  MoveL 756 to (-578.4, 950, 50) mm, rotated rx -180 ry 0 rz 90 deg; joints [-3.759, -80.624, 132.574, 175.231, 52.046, -177.063]
  MoveL 757 to (-578.4, 1000, 50) mm, rotated rx -180 ry 0 rz 90 deg; joints [-3.916, -82.713, 135.158, 175.065, 52.548, -176.994]
  MoveL 758 to (-578.4, 1000, -0.5) mm, rotated rx -180 ry 0 rz 90 deg; joints [-3.916, -79.629, 135.588, 175.277, 56.049, -177.358]
  MoveL 759 to (-578.4, 1000, 50) mm, rotated rx -180 ry 0 rz 90 deg; joints [-3.916, -82.713, 135.158, 175.065, 52.548, -176.994]
  MoveL 760 to (-578.4, 1050, 50) mm, rotated rx -180 ry 0 rz 90 deg; joints [-4.087, -84.881, 137.714, 174.876, 52.943, -176.907]
  MoveL 761 to (-578.4, 1050, -0.5) mm, rotated rx 180 ry 0 rz 90 deg; joints [-4.087, -81.618, 138.166, 175.105, 56.644, -177.304]
  MoveL 762 to (-578.4, 1050, 50) mm, rotated rx -180 ry 0 rz 90 deg; joints [-4.087, -84.881, 137.714, 174.876, 52.943, -176.907]
  MoveL 763 to (-578.4, 1100, 50) mm, rotated rx 180 ry 0 rz 90 deg; joints [-4.273, -87.147, 140.242, 174.661, 53.214, -176.797]
  MoveL 764 to (-578.4, 1100, -0.5) mm, rotated rx -180 ry 0 rz 90 deg; joints [-4.273, -83.684, 140.72, 174.91, 57.139, -177.233]
  MoveL 765 to (-578.4, 1100, 50) mm, rotated rx 180 ry 0 rz 90 deg; joints [-4.273, -87.147, 140.242, 174.661, 53.214, -176.797]
  MoveL 766 to (-578.4, 1150, 50) mm, rotated rx 180 ry 0 rz 90 deg; joints [-4.478, -89.533, 142.744, 174.415, 53.341, -176.659]
  MoveL 767 to (-578.4, 1150, -0.5) mm, rotated rx -180 ry 0 rz 90 deg; joints [-4.478, -85.847, 143.251, 174.69, 57.516, -177.142]
  MoveL 768 to (-578.4, 1150, 50) mm, rotated rx 180 ry 0 rz 90 deg; joints [-4.478, -89.533, 142.744, 174.415, 53.341, -176.659]
  MoveL 769 to (-578.4, 1200, 50) mm, rotated rx 180 ry 0 rz 90 deg; joints [-4.702, -92.068, 145.219, 174.131, 53.295, -176.484]
  MoveL 770 to (-578.4, 1200, -0.5) mm, rotated rx -180 ry 0 rz 90 deg; joints [-4.702, -88.13, 145.761, 174.437, 57.753, -177.025]
  MoveL 771 to (-578.4, 1200, 50) mm, rotated rx 180 ry 0 rz 90 deg; joints [-4.702, -92.068, 145.219, 174.131, 53.295, -176.484]
  MoveL 772 to (-578.4, 1250, 50) mm, rotated rx 180 ry 0 rz 90 deg; joints [-4.951, -94.787, 147.667, 173.8, 53.041, -176.263]
  MoveL 773 to (-578.4, 1250, -0.5) mm, rotated rx -180 ry 0 rz 90 deg; joints [-4.951, -90.565, 148.248, 174.148, 57.818, -176.875]
  MoveL 774 to (-578.4, 1250, 50) mm, rotated rx 180 ry 0 rz 90 deg; joints [-4.951, -94.787, 147.667, 173.8, 53.041, -176.263]
  MoveL 775 to (-578.4, 1300, 50) mm, rotated rx 180 ry 0 rz 90 deg; joints [-5.227, -97.739, 150.087, 173.409, 52.531, -175.979]
  MoveL 776 to (-578.4, 1300, -0.5) mm, rotated rx 180 ry 0 rz 90 deg; joints [-5.227, -93.195, 150.715, 173.811, 57.672, -176.681]
  MoveL 777 to (-578.4, 1300, 50) mm, rotated rx 180 ry 0 rz 90 deg; joints [-5.227, -97.739, 150.087, 173.409, 52.531, -175.979]
  MoveL 778 to (-578.4, 1350, 50) mm, rotated rx 180 ry 0 rz 90 deg; joints [-5.535, -100.986, 152.476, 172.94, 51.702, -175.611]
  MoveL 779 to (-578.4, 1350, -0.5) mm, rotated rx -180 ry 0 rz 90 deg; joints [-5.535, -96.076, 153.16, 173.415, 57.257, -176.427]
  MoveL 780 to (-578.4, 1350, 50) mm, rotated rx 180 ry 0 rz 90 deg; joints [-5.535, -100.986, 152.476, 172.94, 51.702, -175.611]
  MoveL 781 to (-578.4, 1400, 50) mm, rotated rx 180 ry 0 rz 90 deg; joints [-5.882, -104.615, 154.831, 172.364, 50.467, -175.122]
  MoveL 782 to (-578.4, 1400, -0.5) mm, rotated rx -180 ry 0 rz 70 deg; joints [-12.877, -96.991, 153.881, 142.344, 62.693, -160.506]
  MoveL 783 to (-578.4, 1400, 50) mm, rotated rx 180 ry 0 rz 90 deg; joints [-5.882, -104.615, 154.831, 172.364, 50.467, -175.122]
  MoveL 784 to (-578.4, 1450, 50) mm, rotated rx -180 ry 0 rz 50 deg; joints [-18.777, -100.129, 151.872, 115.454, 71.278, -146.007]
  MoveL 785 to (-578.4, 1450, -0.5) mm, rotated rx 180 ry 0 rz 50 deg; joints [-18.777, -95.317, 152.541, 117.006, 73.703, -151.163]
  MoveL 786 to (-578.4, 1450, 50) mm, rotated rx -180 ry 0 rz 50 deg; joints [-18.777, -100.129, 151.872, 115.454, 71.278, -146.007]
  MoveL 787 to (-514.2, 300, 50) mm, rotated rx -180 ry 0 rz 90 deg; joints [-4.407, -56.021, 95.158, 173.039, 39.345, -174.606]
  MoveL 788 to (-514.2, 300, -0.5) mm, rotated rx -180 ry 0 rz 90 deg; joints [-4.407, -54.32, 95.452, 173.318, 41.325, -174.972]
  MoveL 789 to (-514.2, 300, 50) mm, rotated rx -180 ry 0 rz 90 deg; joints [-4.407, -56.021, 95.158, 173.039, 39.345, -174.606]
  MoveL 790 to (-514.2, 650, 50) mm, rotated rx -180 ry 0 rz 90 deg; joints [-5.401, -68.907, 116.122, 172.659, 47.45, -175.021]
  MoveL 791 to (-514.2, 650, -0.5) mm, rotated rx 180 ry 0 rz 90 deg; joints [-5.401, -66.704, 116.453, 172.938, 49.963, -175.444]
  MoveL 792 to (-514.2, 650, 50) mm, rotated rx -180 ry 0 rz 90 deg; joints [-5.401, -68.907, 116.122, 172.659, 47.45, -175.021]
  MoveL 793 to (-476, 230, 50) mm, rotated rx -180 ry 0 rz 90 deg; joints [-5.358, -53.228, 90.342, 171.166, 37.444, -172.965]
  MoveL 794 to (-476, 230, -0.5) mm, rotated rx 180 ry 0 rz 90 deg; joints [-5.358, -51.608, 90.634, 171.529, 39.333, -173.429]
  MoveL 795 to (-476, 230, 50) mm, rotated rx -180 ry 0 rz 90 deg; joints [-5.358, -53.228, 90.342, 171.166, 37.444, -172.965]
  MoveL 796 to (-514.2, 230, 50) mm, rotated rx 180 ry 0 rz 90 deg; joints [-4.25, -53.352, 90.557, 172.994, 37.412, -174.425]
  MoveL 797 to (-514.2, 230, -0.5) mm, rotated rx 180 ry 0 rz 90 deg; joints [-4.25, -51.729, 90.849, 173.283, 39.314, -174.793]
  MoveL 798 to (-514.2, 230, 50) mm, rotated rx 180 ry 0 rz 90 deg; joints [-4.25, -53.352, 90.557, 172.994, 37.412, -174.425]
  MoveL 799 to (-552.4, 230, 50) mm, rotated rx -180 ry 0 rz 90 deg; joints [-3.139, -53.447, 90.723, 174.826, 37.388, -175.885]
  MoveL 800 to (-552.4, 230, -0.5) mm, rotated rx -180 ry 0 rz 90 deg; joints [-3.139, -51.821, 91.014, 175.04, 39.298, -176.158]
  MoveL 801 to (-552.4, 230, 50) mm, rotated rx -180 ry 0 rz 90 deg; joints [-3.139, -53.447, 90.723, 174.826, 37.388, -175.885]
  MoveL 802 to (-476, 420, 50) mm, rotated rx -180 ry 0 rz 90 deg; joints [-5.928, -60.356, 102.467, 171.198, 42.448, -173.481]
  MoveL 803 to (-476, 420, -0.5) mm, rotated rx -180 ry 0 rz 90 deg; joints [-5.928, -58.514, 102.768, 171.537, 44.568, -173.949]
  MoveL 804 to (-476, 420, 50) mm, rotated rx -180 ry 0 rz 90 deg; joints [-5.928, -60.356, 102.467, 171.198, 42.448, -173.481]
  MoveL 805 to (-514.2, 420, 50) mm, rotated rx -180 ry 0 rz 90 deg; joints [-4.704, -60.487, 102.684, 173.016, 42.409, -174.832]
  MoveL 806 to (-514.2, 420, -0.5) mm, rotated rx 180 ry 0 rz 90 deg; joints [-4.704, -58.64, 102.985, 173.286, 44.542, -175.204]
  MoveL 807 to (-514.2, 420, 50) mm, rotated rx -180 ry 0 rz 90 deg; joints [-4.704, -60.487, 102.684, 173.016, 42.409, -174.832]
  MoveL 808 to (-552.4, 420, 50) mm, rotated rx 180 ry 0 rz 90 deg; joints [-3.475, -60.588, 102.85, 174.841, 42.378, -176.184]
  MoveL 809 to (-552.4, 420, -0.5) mm, rotated rx -180 ry 0 rz 90 deg; joints [-3.475, -58.737, 103.152, 175.041, 44.523, -176.46]
  MoveL 810 to (-552.4, 420, 50) mm, rotated rx 180 ry 0 rz 90 deg; joints [-3.475, -60.588, 102.85, 174.841, 42.378, -176.184]
  MoveL 811 to (-476, 1020, 50) mm, rotated rx -180 ry 0 rz 90 deg; joints [-8.922, -83.074, 135.592, 168.809, 53.048, -173.218]
  MoveL 812 to (-476, 1020, -0.5) mm, rotated rx -180 ry 0 rz 90 deg; joints [-8.922, -79.961, 136.026, 169.285, 56.53, -174.042]
  MoveL 813 to (-476, 1020, 50) mm, rotated rx -180 ry 0 rz 90 deg; joints [-8.922, -83.074, 135.592, 168.809, 53.048, -173.218]
  MoveL 814 to (-514.2, 1020, 50) mm, rotated rx -180 ry 0 rz 90 deg; joints [-7.091, -83.302, 135.865, 171.096, 52.898, -174.601]
  MoveL 815 to (-514.2, 1020, -0.5) mm, rotated rx 180 ry 0 rz 90 deg; joints [-7.091, -80.171, 136.302, 171.479, 56.424, -175.263]
  MoveL 816 to (-514.2, 1020, 50) mm, rotated rx -180 ry 0 rz 90 deg; joints [-7.091, -83.302, 135.865, 171.096, 52.898, -174.601]
  MoveL 817 to (-552.4, 1020, 50) mm, rotated rx -180 ry 0 rz 90 deg; joints [-5.246, -83.479, 136.076, 173.407, 52.78, -176.001]
  MoveL 818 to (-552.4, 1020, -0.5) mm, rotated rx -180 ry 0 rz 90 deg; joints [-5.246, -80.334, 136.514, 173.694, 56.341, -176.495]
  MoveL 819 to (-552.4, 1020, 50) mm, rotated rx -180 ry 0 rz 90 deg; joints [-5.246, -83.479, 136.076, 173.407, 52.78, -176.001]
  MoveL 820 to (-655, 50, 50) mm, rotated rx -180 ry 0 rz 90 deg; joints [-0.134, -46.338, 78.157, 179.746, 31.82, -179.784]
  MoveL 821 to (-655, 50, -0.5) mm, rotated rx 180 ry 0 rz 90 deg; joints [-0.134, -44.886, 78.453, 179.758, 33.567, -179.798]
  MoveL 822 to (-655, 50, 50) mm, rotated rx -180 ry 0 rz 90 deg; joints [-0.134, -46.338, 78.157, 179.746, 31.82, -179.784]
  MoveL 823 to (-655, 100, 50) mm, rotated rx 180 ry 0 rz 90 deg; joints [-0.137, -48.409, 81.86, 179.752, 33.452, -179.793]
  MoveL 824 to (-655, 100, -0.5) mm, rotated rx -180 ry 0 rz 90 deg; joints [-0.137, -46.911, 82.153, 179.763, 35.243, -179.806]
  MoveL 825 to (-655, 100, 50) mm, rotated rx 180 ry 0 rz 90 deg; joints [-0.137, -48.409, 81.86, 179.752, 33.452, -179.793]
  MoveL 826 to (-655, 150, 50) mm, rotated rx -180 ry 0 rz 90 deg; joints [-0.14, -50.425, 85.434, 179.755, 35.009, -179.8]
  MoveL 827 to (-655, 150, -0.5) mm, rotated rx 180 ry 0 rz 90 deg; joints [-0.14, -48.879, 85.726, 179.766, 36.847, -179.813]
  MoveL 828 to (-655, 150, 50) mm, rotated rx -180 ry 0 rz 90 deg; joints [-0.14, -50.425, 85.434, 179.755, 35.009, -179.8]
  MoveL 829 to (-655, 200, 50) mm, rotated rx 180 ry 0 rz 90 deg; joints [-0.144, -52.397, 88.893, 179.758, 36.497, -179.806]
  MoveL 830 to (-655, 200, -0.5) mm, rotated rx -180 ry 0 rz 90 deg; joints [-0.144, -50.799, 89.185, 179.768, 38.386, -179.818]
  MoveL 831 to (-655, 200, 50) mm, rotated rx 180 ry 0 rz 90 deg; joints [-0.144, -52.397, 88.893, 179.758, 36.497, -179.806]
  MoveL 832 to (-655, 250, 50) mm, rotated rx 180 ry 0 rz 90 deg; joints [-0.148, -54.33, 92.252, 179.76, 37.922, -179.811]
  MoveL 833 to (-655, 250, -0.5) mm, rotated rx 180 ry 0 rz 90 deg; joints [-0.148, -52.679, 92.544, 179.77, 39.865, -179.823]
  MoveL 834 to (-655, 250, 50) mm, rotated rx 180 ry 0 rz 90 deg; joints [-0.148, -54.33, 92.252, 179.76, 37.922, -179.811]
  MoveL 835 to (-655, 300, 50) mm, rotated rx -180 ry 0 rz 90 deg; joints [-0.151, -56.232, 95.52, 179.761, 39.288, -179.815]
  MoveL 836 to (-655, 300, -0.5) mm, rotated rx 180 ry 0 rz 90 deg; joints [-0.151, -54.526, 95.814, 179.771, 41.289, -179.828]
  MoveL 837 to (-655, 300, 50) mm, rotated rx -180 ry 0 rz 90 deg; joints [-0.151, -56.232, 95.52, 179.761, 39.288, -179.815]
  MoveL 838 to (-655, 350, 50) mm, rotated rx 180 ry 0 rz 90 deg; joints [-0.156, -58.11, 98.708, 179.761, 40.598, -179.819]
  MoveL 839 to (-655, 350, -0.5) mm, rotated rx 180 ry 0 rz 90 deg; joints [-0.156, -56.344, 99.005, 179.77, 42.661, -179.831]
  MoveL 840 to (-655, 350, 50) mm, rotated rx 180 ry 0 rz 90 deg; joints [-0.156, -58.11, 98.708, 179.761, 40.598, -179.819]
  MoveL 841 to (-655, 400, 50) mm, rotated rx 180 ry 0 rz 90 deg; joints [-0.16, -59.969, 101.822, 179.76, 41.854, -179.822]
  MoveL 842 to (-655, 400, -0.5) mm, rotated rx -180 ry 0 rz 90 deg; joints [-0.16, -58.14, 102.123, 179.77, 43.983, -179.834]
  MoveL 843 to (-655, 400, 50) mm, rotated rx 180 ry 0 rz 90 deg; joints [-0.16, -59.969, 101.822, 179.76, 41.854, -179.822]
  MoveL 844 to (-655, 450, 50) mm, rotated rx 180 ry 0 rz 90 deg; joints [-0.164, -61.814, 104.871, 179.759, 43.057, -179.824]
  MoveL 845 to (-655, 450, -0.5) mm, rotated rx -180 ry 0 rz 90 deg; joints [-0.164, -59.918, 105.176, 179.768, 45.258, -179.837]
  MoveL 846 to (-655, 450, 50) mm, rotated rx 180 ry 0 rz 90 deg; joints [-0.164, -61.814, 104.871, 179.759, 43.057, -179.824]
  MoveL 847 to (-655, 500, 50) mm, rotated rx 180 ry 0 rz 90 deg; joints [-0.169, -63.65, 107.859, 179.757, 44.209, -179.826]
  MoveL 848 to (-655, 500, -0.5) mm, rotated rx -180 ry 0 rz 90 deg; joints [-0.169, -61.683, 108.169, 179.767, 46.487, -179.839]
  MoveL 849 to (-655, 500, 50) mm, rotated rx 180 ry 0 rz 90 deg; joints [-0.169, -63.65, 107.859, 179.757, 44.209, -179.826]
  MoveL 850 to (-655, 550, 50) mm, rotated rx 180 ry 0 rz 90 deg; joints [-0.174, -65.483, 110.791, 179.755, 45.309, -179.827]
  MoveL 851 to (-655, 550, -0.5) mm, rotated rx 180 ry 0 rz 90 deg; joints [-0.174, -63.439, 111.108, 179.764, 47.669, -179.841]
  MoveL 852 to (-655, 550, 50) mm, rotated rx 180 ry 0 rz 90 deg; joints [-0.174, -65.483, 110.791, 179.755, 45.309, -179.827]
  MoveL 853 to (-655, 600, 50) mm, rotated rx -180 ry 0 rz 90 deg; joints [-0.18, -67.318, 113.673, 179.751, 46.356, -179.828]
  MoveL 854 to (-655, 600, -0.5) mm, rotated rx 180 ry 0 rz 90 deg; joints [-0.18, -65.192, 113.997, 179.761, 48.806, -179.842]
  MoveL 855 to (-655, 600, 50) mm, rotated rx -180 ry 0 rz 90 deg; joints [-0.18, -67.318, 113.673, 179.751, 46.356, -179.828]
  MoveL 856 to (-655, 650, 50) mm, rotated rx 180 ry 0 rz 90 deg; joints [-0.186, -69.16, 116.509, 179.747, 47.349, -179.829]
  MoveL 857 to (-655, 650, -0.5) mm, rotated rx 180 ry 0 rz 90 deg; joints [-0.186, -66.946, 116.841, 179.757, 49.896, -179.844]
  MoveL 858 to (-655, 650, 50) mm, rotated rx 180 ry 0 rz 90 deg; joints [-0.186, -69.16, 116.509, 179.747, 47.349, -179.829]
  MoveL 859 to (-655, 700, 50) mm, rotated rx 180 ry 0 rz 90 deg; joints [-0.192, -71.015, 119.301, 179.743, 48.286, -179.829]
  MoveL 860 to (-655, 700, -0.5) mm, rotated rx -180 ry 0 rz 90 deg; joints [-0.192, -68.705, 119.643, 179.753, 50.938, -179.844]
  MoveL 861 to (-655, 700, 50) mm, rotated rx 180 ry 0 rz 90 deg; joints [-0.192, -71.015, 119.301, 179.743, 48.286, -179.829]
  MoveL 862 to (-655, 750, 50) mm, rotated rx 180 ry 0 rz 90 deg; joints [-0.199, -72.89, 122.053, 179.737, 49.164, -179.828]
  MoveL 863 to (-655, 750, -0.5) mm, rotated rx 180 ry 0 rz 90 deg; joints [-0.199, -70.476, 122.406, 179.748, 51.929, -179.844]
  MoveL 864 to (-655, 750, 50) mm, rotated rx 180 ry 0 rz 90 deg; joints [-0.199, -72.89, 122.053, 179.737, 49.164, -179.828]
  MoveL 865 to (-655, 800, 50) mm, rotated rx -180 ry 0 rz 90 deg; joints [-0.206, -74.79, 124.768, 179.731, 49.978, -179.827]
  MoveL 866 to (-655, 800, -0.5) mm, rotated rx -180 ry 0 rz 90 deg; joints [-0.206, -72.265, 125.133, 179.742, 52.868, -179.844]
  MoveL 867 to (-655, 800, 50) mm, rotated rx -180 ry 0 rz 90 deg; joints [-0.206, -74.79, 124.768, 179.731, 49.978, -179.827]
  MoveL 868 to (-655, 850, 50) mm, rotated rx -180 ry 0 rz 90 deg; joints [-0.213, -76.725, 127.448, 179.724, 50.724, -179.825]
  MoveL 869 to (-655, 850, -0.5) mm, rotated rx -180 ry 0 rz 90 deg; joints [-0.213, -74.077, 127.827, 179.735, 53.75, -179.843]
  MoveL 870 to (-655, 850, 50) mm, rotated rx -180 ry 0 rz 90 deg; joints [-0.213, -76.725, 127.448, 179.724, 50.724, -179.825]
  MoveL 871 to (-655, 900, 50) mm, rotated rx -180 ry 0 rz 90 deg; joints [-0.222, -78.703, 130.096, 179.716, 51.394, -179.823]
  MoveL 872 to (-655, 900, -0.5) mm, rotated rx 180 ry 0 rz 90 deg; joints [-0.222, -75.92, 130.49, 179.728, 54.57, -179.842]
  MoveL 873 to (-655, 900, 50) mm, rotated rx -180 ry 0 rz 90 deg; joints [-0.222, -78.703, 130.096, 179.716, 51.394, -179.823]
  MoveL 874 to (-655, 950, 50) mm, rotated rx 180 ry 0 rz 90 deg; joints [-0.231, -80.734, 132.713, 179.707, 51.979, -179.82]
  MoveL 875 to (-655, 950, -0.5) mm, rotated rx 180 ry 0 rz 90 deg; joints [-0.231, -77.804, 133.125, 179.72, 55.321, -179.84]
  MoveL 876 to (-655, 950, 50) mm, rotated rx 180 ry 0 rz 90 deg; joints [-0.231, -80.734, 132.713, 179.707, 51.979, -179.82]
  MoveL 877 to (-655, 1000, 50) mm, rotated rx -180 ry 0 rz 90 deg; joints [-0.24, -82.832, 135.301, 179.697, 52.47, -179.815]
  MoveL 878 to (-655, 1000, -0.5) mm, rotated rx 180 ry 0 rz 90 deg; joints [-0.24, -79.738, 135.732, 179.71, 55.994, -179.838]
  MoveL 879 to (-655, 1000, 50) mm, rotated rx -180 ry 0 rz 90 deg; joints [-0.24, -82.832, 135.301, 179.697, 52.47, -179.815]
  MoveL 880 to (-655, 1050, 50) mm, rotated rx 180 ry 0 rz 90 deg; joints [-0.251, -85.01, 137.861, 179.685, 52.851, -179.81]
  MoveL 881 to (-655, 1050, -0.5) mm, rotated rx -180 ry 0 rz 90 deg; joints [-0.251, -81.736, 138.315, 179.699, 56.58, -179.834]
  MoveL 882 to (-655, 1050, 50) mm, rotated rx 180 ry 0 rz 90 deg; joints [-0.251, -85.01, 137.861, 179.685, 52.851, -179.81]
  MoveL 883 to (-655, 1100, 50) mm, rotated rx 180 ry 0 rz 90 deg; joints [-0.262, -87.289, 140.395, 179.672, 53.107, -179.803]
  MoveL 884 to (-655, 1100, -0.5) mm, rotated rx 180 ry 0 rz 90 deg; joints [-0.262, -83.813, 140.875, 179.687, 57.062, -179.83]
  MoveL 885 to (-655, 1100, 50) mm, rotated rx 180 ry 0 rz 90 deg; joints [-0.262, -87.289, 140.395, 179.672, 53.107, -179.803]
  MoveL 886 to (-655, 1150, 50) mm, rotated rx 180 ry 0 rz 90 deg; joints [-0.275, -89.69, 142.902, 179.657, 53.213, -179.794]
  MoveL 887 to (-655, 1150, -0.5) mm, rotated rx -180 ry 0 rz 90 deg; joints [-0.275, -85.989, 143.412, 179.674, 57.424, -179.824]
  MoveL 888 to (-655, 1150, 50) mm, rotated rx 180 ry 0 rz 90 deg; joints [-0.275, -89.69, 142.902, 179.657, 53.213, -179.794]
  MoveL 889 to (-655, 1200, 50) mm, rotated rx -180 ry 0 rz 90 deg; joints [-0.289, -92.243, 145.383, 179.639, 53.141, -179.783]
  MoveL 890 to (-655, 1200, -0.5) mm, rotated rx 180 ry 0 rz 90 deg; joints [-0.289, -88.288, 145.928, 179.658, 57.64, -179.817]
  MoveL 891 to (-655, 1200, 50) mm, rotated rx -180 ry 0 rz 90 deg; joints [-0.289, -92.243, 145.383, 179.639, 53.141, -179.783]
  MoveL 892 to (-655, 1250, 50) mm, rotated rx -180 ry 0 rz 90 deg; joints [-0.304, -94.987, 147.838, 179.618, 52.852, -179.77]
  MoveL 893 to (-655, 1250, -0.5) mm, rotated rx -180 ry 0 rz 90 deg; joints [-0.304, -90.744, 148.423, 179.64, 57.68, -179.808]
  MoveL 894 to (-655, 1250, 50) mm, rotated rx -180 ry 0 rz 90 deg; joints [-0.304, -94.987, 147.838, 179.618, 52.852, -179.77]
  MoveL 895 to (-783.4, 50, 50) mm, rotated rx 180 ry 0 rz 90 deg; joints [3.297, -46.188, 77.889, 186.256, 31.854, -185.32]
  MoveL 896 to (-783.4, 50, -0.5) mm, rotated rx 180 ry 0 rz 90 deg; joints [3.297, -44.74, 78.185, 185.967, 33.588, -184.977]
  MoveL 897 to (-783.4, 50, 50) mm, rotated rx 180 ry 0 rz 90 deg; joints [3.297, -46.188, 77.889, 186.256, 31.854, -185.32]
  MoveL 898 to (-783.4, 100, 50) mm, rotated rx -180 ry 0 rz 90 deg; joints [3.376, -48.26, 81.596, 186.127, 33.486, -185.116]
  MoveL 899 to (-783.4, 100, -0.5) mm, rotated rx 180 ry 0 rz 90 deg; joints [3.376, -46.766, 81.889, 185.854, 35.265, -184.785]
  MoveL 900 to (-783.4, 100, 50) mm, rotated rx -180 ry 0 rz 90 deg; joints [3.376, -48.26, 81.596, 186.127, 33.486, -185.116]
  MoveL 901 to (-783.4, 150, 50) mm, rotated rx 180 ry 0 rz 90 deg; joints [3.458, -50.277, 85.172, 186.03, 35.044, -184.943]
  MoveL 902 to (-783.4, 150, -0.5) mm, rotated rx 180 ry 0 rz 90 deg; joints [3.458, -48.734, 85.464, 185.77, 36.869, -184.622]
  MoveL 903 to (-783.4, 150, 50) mm, rotated rx 180 ry 0 rz 90 deg; joints [3.458, -50.277, 85.172, 186.03, 35.044, -184.943]
  MoveL 904 to (-783.4, 200, 50) mm, rotated rx 180 ry 0 rz 90 deg; joints [3.545, -52.248, 88.633, 185.962, 36.534, -184.796]
  MoveL 905 to (-783.4, 200, -0.5) mm, rotated rx -180 ry 0 rz 90 deg; joints [3.545, -50.654, 88.925, 185.712, 38.409, -184.481]
  MoveL 906 to (-783.4, 200, 50) mm, rotated rx 180 ry 0 rz 90 deg; joints [3.545, -52.248, 88.633, 185.962, 36.534, -184.796]
  MoveL 907 to (-783.4, 250, 50) mm, rotated rx -180 ry 0 rz 90 deg; joints [3.636, -54.18, 91.992, 185.917, 37.961, -184.672]
  MoveL 908 to (-783.4, 250, -0.5) mm, rotated rx -180 ry 0 rz 90 deg; joints [3.636, -52.534, 92.285, 185.675, 39.89, -184.36]
  MoveL 909 to (-783.4, 250, 50) mm, rotated rx -180 ry 0 rz 90 deg; joints [3.636, -54.18, 91.992, 185.917, 37.961, -184.672]
  MoveL 910 to (-783.4, 300, 50) mm, rotated rx 180 ry 0 rz 90 deg; joints [3.732, -56.081, 95.261, 185.894, 39.329, -184.566]
  MoveL 911 to (-783.4, 300, -0.5) mm, rotated rx -180 ry 0 rz 90 deg; joints [3.732, -54.379, 95.555, 185.658, 41.315, -184.255]
  MoveL 912 to (-783.4, 300, 50) mm, rotated rx 180 ry 0 rz 90 deg; joints [3.732, -56.081, 95.261, 185.894, 39.329, -184.566]
  MoveL 913 to (-783.4, 350, 50) mm, rotated rx 180 ry 0 rz 90 deg; joints [3.833, -57.956, 98.448, 185.89, 40.642, -184.476]
  MoveL 914 to (-783.4, 350, -0.5) mm, rotated rx 180 ry 0 rz 90 deg; joints [3.833, -56.195, 98.745, 185.658, 42.689, -184.165]
  MoveL 915 to (-783.4, 350, 50) mm, rotated rx 180 ry 0 rz 90 deg; joints [3.833, -57.956, 98.448, 185.89, 40.642, -184.476]
  MoveL 916 to (-783.4, 400, 50) mm, rotated rx -180 ry 0 rz 90 deg; joints [3.939, -59.812, 101.561, 185.904, 41.901, -184.402]
  MoveL 917 to (-783.4, 400, -0.5) mm, rotated rx -180 ry 0 rz 90 deg; joints [3.939, -57.988, 101.861, 185.674, 44.014, -184.087]
  MoveL 918 to (-783.4, 400, 50) mm, rotated rx -180 ry 0 rz 90 deg; joints [3.939, -59.812, 101.561, 185.904, 41.901, -184.402]
  MoveL 919 to (-783.4, 450, 50) mm, rotated rx 180 ry 0 rz 90 deg; joints [4.052, -61.653, 104.608, 185.935, 43.108, -184.34]
  MoveL 920 to (-783.4, 450, -0.5) mm, rotated rx 180 ry 0 rz 90 deg; joints [4.052, -59.763, 104.912, 185.706, 45.291, -184.021]
  MoveL 921 to (-783.4, 450, 50) mm, rotated rx 180 ry 0 rz 90 deg; joints [4.052, -61.653, 104.608, 185.935, 43.108, -184.34]
  MoveL 922 to (-783.4, 500, 50) mm, rotated rx 180 ry 0 rz 90 deg; joints [4.171, -63.486, 107.593, 185.982, 44.264, -184.291]
  MoveL 923 to (-783.4, 500, -0.5) mm, rotated rx -180 ry 0 rz 90 deg; joints [4.171, -61.525, 107.903, 185.753, 46.523, -183.965]
  MoveL 924 to (-783.4, 500, 50) mm, rotated rx 180 ry 0 rz 90 deg; joints [4.171, -63.486, 107.593, 185.982, 44.264, -184.291]
  MoveL 925 to (-783.4, 550, 50) mm, rotated rx -180 ry 0 rz 90 deg; joints [4.298, -65.314, 110.523, 186.045, 45.368, -184.255]
  MoveL 926 to (-783.4, 550, -0.5) mm, rotated rx 180 ry 0 rz 90 deg; joints [4.298, -63.277, 110.838, 185.815, 47.709, -183.92]
  MoveL 927 to (-783.4, 550, 50) mm, rotated rx -180 ry 0 rz 90 deg; joints [4.298, -65.314, 110.523, 186.045, 45.368, -184.255]
  MoveL 928 to (-783.4, 600, 50) mm, rotated rx -180 ry 0 rz 90 deg; joints [4.432, -67.143, 113.401, 186.124, 46.422, -184.23]
  MoveL 929 to (-783.4, 600, -0.5) mm, rotated rx -180 ry 0 rz 90 deg; joints [4.432, -65.025, 113.724, 185.891, 48.849, -183.884]
  MoveL 930 to (-783.4, 600, 50) mm, rotated rx -180 ry 0 rz 90 deg; joints [4.432, -67.143, 113.401, 186.124, 46.422, -184.23]
  MoveL 931 to (-783.4, 650, 50) mm, rotated rx -180 ry 0 rz 90 deg; joints [4.575, -68.978, 116.232, 186.219, 47.422, -184.217]
  MoveL 932 to (-783.4, 650, -0.5) mm, rotated rx -180 ry 0 rz 90 deg; joints [4.575, -66.773, 116.563, 185.982, 49.944, -183.858]
  MoveL 933 to (-783.4, 650, 50) mm, rotated rx -180 ry 0 rz 90 deg; joints [4.575, -68.978, 116.232, 186.219, 47.422, -184.217]
  MoveL 934 to (-783.4, 700, 50) mm, rotated rx -180 ry 0 rz 90 deg; joints [4.728, -70.826, 119.019, 186.332, 48.367, -184.216]
  MoveL 935 to (-783.4, 700, -0.5) mm, rotated rx -180 ry 0 rz 90 deg; joints [4.728, -68.526, 119.359, 186.089, 50.992, -183.841]
  MoveL 936 to (-783.4, 700, 50) mm, rotated rx -180 ry 0 rz 90 deg; joints [4.728, -70.826, 119.019, 186.332, 48.367, -184.216]
  MoveL 937 to (-783.4, 750, 50) mm, rotated rx -180 ry 0 rz 90 deg; joints [4.891, -72.691, 121.765, 186.462, 49.254, -184.228]
  MoveL 938 to (-783.4, 750, -0.5) mm, rotated rx 180 ry 0 rz 90 deg; joints [4.891, -70.289, 122.117, 186.212, 51.991, -183.835]
  MoveL 939 to (-783.4, 750, 50) mm, rotated rx -180 ry 0 rz 90 deg; joints [4.891, -72.691, 121.765, 186.462, 49.254, -184.228]
  MoveL 940 to (-783.4, 800, 50) mm, rotated rx -180 ry 0 rz 90 deg; joints [5.066, -74.582, 124.474, 186.611, 50.08, -184.254]
  MoveL 941 to (-783.4, 800, -0.5) mm, rotated rx 180 ry 0 rz 90 deg; joints [5.066, -72.069, 124.837, 186.353, 52.938, -183.839]
  MoveL 942 to (-783.4, 800, 50) mm, rotated rx -180 ry 0 rz 90 deg; joints [5.066, -74.582, 124.474, 186.611, 50.08, -184.254]
  MoveL 943 to (-783.4, 850, 50) mm, rotated rx 180 ry 0 rz 90 deg; joints [5.254, -76.504, 127.147, 186.782, 50.84, -184.295]
  MoveL 944 to (-783.4, 850, -0.5) mm, rotated rx -180 ry 0 rz 90 deg; joints [5.254, -73.871, 127.524, 186.513, 53.83, -183.855]
  MoveL 945 to (-783.4, 850, 50) mm, rotated rx 180 ry 0 rz 90 deg; joints [5.254, -76.504, 127.147, 186.782, 50.84, -184.295]
  MoveL 946 to (-783.4, 900, 50) mm, rotated rx -180 ry 0 rz 90 deg; joints [5.456, -78.468, 129.787, 186.975, 51.526, -184.353]
  MoveL 947 to (-783.4, 900, -0.5) mm, rotated rx 180 ry 0 rz 90 deg; joints [5.456, -75.702, 130.179, 186.693, 54.662, -183.883]
  MoveL 948 to (-783.4, 900, 50) mm, rotated rx -180 ry 0 rz 90 deg; joints [5.456, -78.468, 129.787, 186.975, 51.526, -184.353]
  MoveL 949 to (-783.4, 950, 50) mm, rotated rx -180 ry 0 rz 90 deg; joints [5.674, -80.483, 132.395, 187.195, 52.132, -184.431]
  MoveL 950 to (-783.4, 950, -0.5) mm, rotated rx 180 ry 0 rz 90 deg; joints [5.674, -77.572, 132.804, 186.896, 55.427, -183.926]
  MoveL 951 to (-783.4, 950, 50) mm, rotated rx -180 ry 0 rz 90 deg; joints [5.674, -80.483, 132.395, 187.195, 52.132, -184.431]
  MoveL 952 to (-783.4, 1000, 50) mm, rotated rx -180 ry 0 rz 90 deg; joints [5.91, -82.561, 134.973, 187.443, 52.647, -184.532]
  MoveL 953 to (-783.4, 1000, -0.5) mm, rotated rx 180 ry 0 rz 90 deg; joints [5.91, -79.489, 135.402, 187.125, 56.119, -183.986]
  MoveL 954 to (-783.4, 1000, 50) mm, rotated rx -180 ry 0 rz 90 deg; joints [5.91, -82.561, 134.973, 187.443, 52.647, -184.532]
  MoveL 955 to (-783.4, 1050, 50) mm, rotated rx 180 ry 0 rz 90 deg; joints [6.167, -84.716, 137.523, 187.725, 53.058, -184.661]
  MoveL 956 to (-783.4, 1050, -0.5) mm, rotated rx 180 ry 0 rz 90 deg; joints [6.167, -81.467, 137.974, 187.383, 56.726, -184.066]
  MoveL 957 to (-783.4, 1050, 50) mm, rotated rx 180 ry 0 rz 90 deg; joints [6.167, -84.716, 137.523, 187.725, 53.058, -184.661]
  MoveL 958 to (-783.4, 1100, 50) mm, rotated rx -180 ry 0 rz 90 deg; joints [6.447, -86.966, 140.045, 188.045, 53.351, -184.823]
  MoveL 959 to (-783.4, 1100, -0.5) mm, rotated rx 180 ry 0 rz 90 deg; joints [6.447, -83.519, 140.521, 187.674, 57.237, -184.17]
  MoveL 960 to (-783.4, 1100, 50) mm, rotated rx -180 ry 0 rz 90 deg; joints [6.447, -86.966, 140.045, 188.045, 53.351, -184.823]
  MoveL 961 to (-783.4, 1150, 50) mm, rotated rx -180 ry 0 rz 90 deg; joints [6.754, -89.332, 142.539, 188.412, 53.504, -185.027]
  MoveL 962 to (-783.4, 1150, -0.5) mm, rotated rx -180 ry 0 rz 90 deg; joints [6.754, -85.665, 143.044, 188.004, 57.633, -184.305]
  MoveL 963 to (-783.4, 1150, 50) mm, rotated rx -180 ry 0 rz 90 deg; joints [6.754, -89.332, 142.539, 188.412, 53.504, -185.027]
  MoveL 964 to (-783.4, 1200, 50) mm, rotated rx 180 ry 0 rz 90 deg; joints [7.091, -91.842, 145.006, 188.835, 53.491, -185.283]
  MoveL 965 to (-783.4, 1200, -0.5) mm, rotated rx -180 ry 0 rz 90 deg; joints [7.091, -87.928, 145.545, 188.38, 57.895, -184.476]
  MoveL 966 to (-783.4, 1200, 50) mm, rotated rx 180 ry 0 rz 90 deg; joints [7.091, -91.842, 145.006, 188.835, 53.491, -185.283]
  MoveL 967 to (-783.4, 1250, 50) mm, rotated rx -180 ry 0 rz 90 deg; joints [7.463, -94.531, 147.446, 189.325, 53.28, -185.607]
  MoveL 968 to (-783.4, 1250, -0.5) mm, rotated rx 180 ry 0 rz 90 deg; joints [7.463, -90.337, 148.023, 188.811, 57.993, -184.697]
  MoveL 969 to (-783.4, 1250, 50) mm, rotated rx -180 ry 0 rz 90 deg; joints [7.463, -94.531, 147.446, 189.325, 53.28, -185.607]
  MoveL 970 to (-719.2, 300, 50) mm, rotated rx 180 ry 0 rz 90 deg; joints [1.792, -56.198, 95.461, 182.83, 39.298, -182.191]
  MoveL 971 to (-719.2, 300, -0.5) mm, rotated rx 180 ry 0 rz 90 deg; joints [1.792, -54.492, 95.755, 182.716, 41.295, -182.041]
  MoveL 972 to (-719.2, 300, 50) mm, rotated rx 180 ry 0 rz 90 deg; joints [1.792, -56.198, 95.461, 182.83, 39.298, -182.191]
  MoveL 973 to (-719.2, 650, 50) mm, rotated rx -180 ry 0 rz 90 deg; joints [2.199, -69.119, 116.445, 182.989, 47.366, -182.026]
  MoveL 974 to (-719.2, 650, -0.5) mm, rotated rx -180 ry 0 rz 90 deg; joints [2.199, -66.906, 116.777, 182.874, 49.907, -181.852]
  MoveL 975 to (-719.2, 650, 50) mm, rotated rx -180 ry 0 rz 90 deg; joints [2.199, -69.119, 116.445, 182.989, 47.366, -182.026]
  MoveL 976 to (-681, 230, 50) mm, rotated rx -180 ry 0 rz 90 deg; joints [0.613, -53.557, 90.913, 181.011, 37.36, -180.803]
  MoveL 977 to (-681, 230, -0.5) mm, rotated rx 180 ry 0 rz 90 deg; joints [0.613, -51.928, 91.205, 180.969, 39.281, -180.75]
  MoveL 978 to (-681, 230, 50) mm, rotated rx -180 ry 0 rz 90 deg; joints [0.613, -53.557, 90.913, 181.011, 37.36, -180.803]
  MoveL 979 to (-719.2, 230, 50) mm, rotated rx 180 ry 0 rz 90 deg; joints [1.728, -53.526, 90.86, 182.848, 37.368, -182.264]
  MoveL 980 to (-719.2, 230, -0.5) mm, rotated rx -180 ry 0 rz 90 deg; joints [1.728, -51.898, 91.152, 182.73, 39.286, -182.114]
  MoveL 981 to (-719.2, 230, 50) mm, rotated rx 180 ry 0 rz 90 deg; joints [1.728, -53.526, 90.86, 182.848, 37.368, -182.264]
  MoveL 982 to (-757.4, 230, 50) mm, rotated rx -180 ry 0 rz 90 deg; joints [2.842, -53.468, 90.758, 184.684, 37.383, -183.725]
  MoveL 983 to (-757.4, 230, -0.5) mm, rotated rx -180 ry 0 rz 90 deg; joints [2.842, -51.841, 91.05, 184.49, 39.295, -183.478]
  MoveL 984 to (-757.4, 230, 50) mm, rotated rx -180 ry 0 rz 90 deg; joints [2.842, -53.468, 90.758, 184.684, 37.383, -183.725]
  MoveL 985 to (-681, 420, 50) mm, rotated rx 180 ry 0 rz 90 deg; joints [0.679, -60.704, 103.042, 181.008, 42.343, -180.745]
  MoveL 986 to (-681, 420, -0.5) mm, rotated rx 180 ry 0 rz 90 deg; joints [0.679, -58.849, 103.344, 180.969, 44.5, -180.691]
  MoveL 987 to (-681, 420, 50) mm, rotated rx 180 ry 0 rz 90 deg; joints [0.679, -60.704, 103.042, 181.008, 42.343, -180.745]
  MoveL 988 to (-719.2, 420, 50) mm, rotated rx 180 ry 0 rz 90 deg; joints [1.913, -60.672, 102.989, 182.841, 42.353, -182.1]
  MoveL 989 to (-719.2, 420, -0.5) mm, rotated rx 180 ry 0 rz 90 deg; joints [1.913, -58.818, 103.291, 182.73, 44.506, -181.948]
  MoveL 990 to (-719.2, 420, 50) mm, rotated rx 180 ry 0 rz 90 deg; joints [1.913, -60.672, 102.989, 182.841, 42.353, -182.1]
  MoveL 991 to (-757.4, 420, 50) mm, rotated rx -180 ry 0 rz 90 deg; joints [3.146, -60.61, 102.886, 184.671, 42.372, -183.454]
  MoveL 992 to (-757.4, 420, -0.5) mm, rotated rx 180 ry 0 rz 90 deg; joints [3.146, -58.758, 103.188, 184.49, 44.518, -183.204]
  MoveL 993 to (-757.4, 420, 50) mm, rotated rx -180 ry 0 rz 90 deg; joints [3.146, -60.61, 102.886, 184.671, 42.372, -183.454]
  MoveL 994 to (-681, 1020, 50) mm, rotated rx -180 ry 0 rz 90 deg; joints [1.027, -83.685, 136.319, 181.291, 52.642, -180.784]
  MoveL 995 to (-681, 1020, -0.5) mm, rotated rx -180 ry 0 rz 90 deg; joints [1.027, -80.522, 136.759, 181.235, 56.243, -180.686]
  MoveL 996 to (-681, 1020, 50) mm, rotated rx -180 ry 0 rz 90 deg; joints [1.027, -83.685, 136.319, 181.291, 52.642, -180.784]
  MoveL 997 to (-719.2, 1020, 50) mm, rotated rx -180 ry 0 rz 90 deg; joints [2.892, -83.628, 136.252, 183.637, 52.68, -182.207]
  MoveL 998 to (-719.2, 1020, -0.5) mm, rotated rx 180 ry 0 rz 90 deg; joints [2.892, -80.47, 136.692, 183.478, 56.27, -181.933]
  MoveL 999 to (-719.2, 1020, 50) mm, rotated rx -180 ry 0 rz 90 deg; joints [2.892, -83.628, 136.252, 183.637, 52.68, -182.207]
  MoveL 1000 to (-757.4, 1020, 50) mm, rotated rx 180 ry 0 rz 90 deg; joints [4.751, -83.518, 136.122, 185.972, 52.754, -183.623]
  MoveL 1001 to (-757.4, 1020, -0.5) mm, rotated rx 180 ry 0 rz 90 deg; joints [4.751, -80.369, 136.56, 185.712, 56.323, -183.174]
  MoveL 1002 to (-757.4, 1020, 50) mm, rotated rx 180 ry 0 rz 90 deg; joints [4.751, -83.518, 136.122, 185.972, 52.754, -183.623]
  MoveL 1003 to (-890, 50, 50) mm, rotated rx 180 ry 0 rz 90 deg; joints [6.129, -45.818, 77.224, 191.643, 31.938, -189.919]
  MoveL 1004 to (-890, 50, -0.5) mm, rotated rx -180 ry 0 rz 90 deg; joints [6.129, -44.378, 77.52, 191.111, 33.641, -189.286]
  MoveL 1005 to (-890, 50, 50) mm, rotated rx 180 ry 0 rz 90 deg; joints [6.129, -45.818, 77.224, 191.643, 31.938, -189.919]
  MoveL 1006 to (-890, 100, 50) mm, rotated rx 180 ry 0 rz 90 deg; joints [6.274, -47.892, 80.94, 191.398, 33.571, -189.535]
  MoveL 1007 to (-890, 100, -0.5) mm, rotated rx 180 ry 0 rz 90 deg; joints [6.274, -46.406, 81.234, 190.897, 35.318, -188.927]
  MoveL 1008 to (-890, 100, 50) mm, rotated rx 180 ry 0 rz 90 deg; joints [6.274, -47.892, 80.94, 191.398, 33.571, -189.535]
  MoveL 1009 to (-890, 150, 50) mm, rotated rx -180 ry 0 rz 90 deg; joints [6.426, -49.91, 84.523, 191.216, 35.131, -189.211]
  MoveL 1010 to (-890, 150, -0.5) mm, rotated rx 180 ry 0 rz 90 deg; joints [6.426, -48.376, 84.815, 190.738, 36.924, -188.62]
  MoveL 1011 to (-890, 150, 50) mm, rotated rx -180 ry 0 rz 90 deg; joints [6.426, -49.91, 84.523, 191.216, 35.131, -189.211]
  MoveL 1012 to (-890, 200, 50) mm, rotated rx 180 ry 0 rz 90 deg; joints [6.586, -51.879, 87.988, 191.085, 36.624, -188.936]
  MoveL 1013 to (-890, 200, -0.5) mm, rotated rx -180 ry 0 rz 90 deg; joints [6.586, -50.295, 88.28, 190.626, 38.466, -188.357]
  MoveL 1014 to (-890, 200, 50) mm, rotated rx 180 ry 0 rz 90 deg; joints [6.586, -51.879, 87.988, 191.085, 36.624, -188.936]
  MoveL 1015 to (-890, 250, 50) mm, rotated rx 180 ry 0 rz 90 deg; joints [6.754, -53.809, 91.35, 190.999, 38.056, -188.701]
  MoveL 1016 to (-890, 250, -0.5) mm, rotated rx -180 ry 0 rz 90 deg; joints [6.754, -52.173, 91.642, 190.554, 39.95, -188.129]
  MoveL 1017 to (-890, 250, 50) mm, rotated rx 180 ry 0 rz 90 deg; joints [6.754, -53.809, 91.35, 190.999, 38.056, -188.701]
  MoveL 1018 to (-890, 300, 50) mm, rotated rx -180 ry 0 rz 90 deg; joints [6.931, -55.705, 94.619, 190.953, 39.429, -188.502]
  MoveL 1019 to (-890, 300, -0.5) mm, rotated rx -180 ry 0 rz 90 deg; joints [6.931, -54.015, 94.912, 190.519, 41.379, -187.932]
  MoveL 1020 to (-890, 300, 50) mm, rotated rx -180 ry 0 rz 90 deg; joints [6.931, -55.705, 94.619, 190.953, 39.429, -188.502]
  MoveL 1021 to (-890, 350, 50) mm, rotated rx -180 ry 0 rz 90 deg; joints [7.117, -57.575, 97.804, 190.942, 40.748, -188.333]
  MoveL 1022 to (-890, 350, -0.5) mm, rotated rx 180 ry 0 rz 90 deg; joints [7.117, -55.827, 98.1, 190.516, 42.757, -187.761]
  MoveL 1023 to (-890, 350, 50) mm, rotated rx -180 ry 0 rz 90 deg; joints [7.117, -57.575, 97.804, 190.942, 40.748, -188.333]
  MoveL 1024 to (-890, 400, 50) mm, rotated rx -180 ry 0 rz 90 deg; joints [7.314, -59.424, 100.914, 190.964, 42.015, -188.191]
  MoveL 1025 to (-890, 400, -0.5) mm, rotated rx -180 ry 0 rz 90 deg; joints [7.314, -57.614, 101.214, 190.543, 44.087, -187.614]
  MoveL 1026 to (-890, 400, 50) mm, rotated rx -180 ry 0 rz 90 deg; joints [7.314, -59.424, 100.914, 190.964, 42.015, -188.191]
  MoveL 1027 to (-890, 450, 50) mm, rotated rx -180 ry 0 rz 90 deg; joints [7.521, -61.257, 103.956, 191.017, 43.23, -188.074]
  MoveL 1028 to (-890, 450, -0.5) mm, rotated rx 180 ry 0 rz 90 deg; joints [7.521, -59.382, 104.26, 190.599, 45.371, -187.489]
  MoveL 1029 to (-890, 450, 50) mm, rotated rx -180 ry 0 rz 90 deg; joints [7.521, -61.257, 103.956, 191.017, 43.23, -188.074]
  MoveL 1030 to (-890, 500, 50) mm, rotated rx -180 ry 0 rz 90 deg; joints [7.741, -63.08, 106.935, 191.1, 44.397, -187.98]
  MoveL 1031 to (-890, 500, -0.5) mm, rotated rx -180 ry 0 rz 90 deg; joints [7.741, -61.135, 107.244, 190.682, 46.609, -187.383]
  MoveL 1032 to (-890, 500, 50) mm, rotated rx -180 ry 0 rz 90 deg; joints [7.741, -63.08, 106.935, 191.1, 44.397, -187.98]
  MoveL 1033 to (-890, 550, 50) mm, rotated rx -180 ry 0 rz 90 deg; joints [7.974, -64.896, 109.857, 191.212, 45.514, -187.908]
  MoveL 1034 to (-890, 550, -0.5) mm, rotated rx 180 ry 0 rz 90 deg; joints [7.974, -62.877, 110.172, 190.792, 47.804, -187.296]
  MoveL 1035 to (-890, 550, 50) mm, rotated rx -180 ry 0 rz 90 deg; joints [7.974, -64.896, 109.857, 191.212, 45.514, -187.908]
  MoveL 1036 to (-890, 600, 50) mm, rotated rx 180 ry 0 rz 90 deg; joints [8.221, -66.711, 112.727, 191.353, 46.581, -187.858]
  MoveL 1037 to (-890, 600, -0.5) mm, rotated rx -180 ry 0 rz 90 deg; joints [8.221, -64.613, 113.048, 190.929, 48.955, -187.226]
  MoveL 1038 to (-890, 600, 50) mm, rotated rx 180 ry 0 rz 90 deg; joints [8.221, -66.711, 112.727, 191.353, 46.581, -187.858]
  MoveL 1039 to (-890, 650, 50) mm, rotated rx -180 ry 0 rz 90 deg; joints [8.484, -68.531, 115.547, 191.524, 47.598, -187.829]
  MoveL 1040 to (-890, 650, -0.5) mm, rotated rx 180 ry 0 rz 90 deg; joints [8.484, -66.347, 115.876, 191.093, 50.062, -187.174]
  MoveL 1041 to (-890, 650, 50) mm, rotated rx -180 ry 0 rz 90 deg; joints [8.484, -68.531, 115.547, 191.524, 47.598, -187.829]
  MoveL 1042 to (-890, 700, 50) mm, rotated rx 180 ry 0 rz 90 deg; joints [8.763, -70.36, 118.322, 191.726, 48.562, -187.821]
  MoveL 1043 to (-890, 700, -0.5) mm, rotated rx -180 ry 0 rz 90 deg; joints [8.763, -68.084, 118.66, 191.286, 51.124, -187.139]
  MoveL 1044 to (-890, 700, 50) mm, rotated rx 180 ry 0 rz 90 deg; joints [8.763, -70.36, 118.322, 191.726, 48.562, -187.821]
  MoveL 1045 to (-890, 750, 50) mm, rotated rx 180 ry 0 rz 90 deg; joints [9.062, -72.204, 121.055, 191.96, 49.473, -187.837]
  MoveL 1046 to (-890, 750, -0.5) mm, rotated rx 180 ry 0 rz 90 deg; joints [9.062, -69.829, 121.403, 191.508, 52.139, -187.123]
  MoveL 1047 to (-890, 750, 50) mm, rotated rx 180 ry 0 rz 90 deg; joints [9.062, -72.204, 121.055, 191.96, 49.473, -187.837]
  MoveL 1048 to (-890, 800, 50) mm, rotated rx 180 ry 0 rz 90 deg; joints [9.382, -74.07, 123.748, 192.228, 50.326, -187.877]
  MoveL 1049 to (-890, 800, -0.5) mm, rotated rx -180 ry 0 rz 90 deg; joints [9.382, -71.588, 124.108, 191.762, 53.106, -187.125]
  MoveL 1050 to (-890, 800, 50) mm, rotated rx 180 ry 0 rz 90 deg; joints [9.382, -74.07, 123.748, 192.228, 50.326, -187.877]
  MoveL 1051 to (-890, 850, 50) mm, rotated rx -180 ry 0 rz 90 deg; joints [9.725, -75.964, 126.404, 192.533, 51.117, -187.944]
  MoveL 1052 to (-890, 850, -0.5) mm, rotated rx 180 ry 0 rz 90 deg; joints [9.725, -73.365, 126.777, 192.049, 54.021, -187.147]
  MoveL 1053 to (-890, 850, 50) mm, rotated rx -180 ry 0 rz 90 deg; joints [9.725, -75.964, 126.404, 192.533, 51.117, -187.944]
  MoveL 1054 to (-890, 900, 50) mm, rotated rx 180 ry 0 rz 90 deg; joints [10.094, -77.894, 129.025, 192.879, 51.842, -188.041]
  MoveL 1055 to (-890, 900, -0.5) mm, rotated rx -180 ry 0 rz 90 deg; joints [10.094, -75.167, 129.412, 192.373, 54.881, -187.193]
  MoveL 1056 to (-890, 900, 50) mm, rotated rx 180 ry 0 rz 90 deg; joints [10.094, -77.894, 129.025, 192.879, 51.842, -188.041]
  MoveL 1057 to (-890, 950, 50) mm, rotated rx -180 ry 0 rz 90 deg; joints [10.491, -79.869, 131.612, 193.27, 52.494, -188.171]
  MoveL 1058 to (-890, 950, -0.5) mm, rotated rx 180 ry 0 rz 90 deg; joints [10.491, -77.003, 132.016, 192.737, 55.68, -187.263]
  MoveL 1059 to (-890, 950, 50) mm, rotated rx -180 ry 0 rz 90 deg; joints [10.491, -79.869, 131.612, 193.27, 52.494, -188.171]
  MoveL 1060 to (-890, 1000, 50) mm, rotated rx 180 ry 0 rz 90 deg; joints [10.921, -81.901, 134.167, 193.711, 53.065, -188.341]
  MoveL 1061 to (-890, 1000, -0.5) mm, rotated rx -180 ry 0 rz 90 deg; joints [10.921, -78.881, 134.589, 193.146, 56.413, -187.362]
  MoveL 1062 to (-890, 1000, 50) mm, rotated rx 180 ry 0 rz 90 deg; joints [10.921, -81.901, 134.167, 193.711, 53.065, -188.341]
  MoveL 1063 to (-890, 1050, 50) mm, rotated rx -180 ry 0 rz 90 deg; joints [11.387, -84, 136.691, 194.209, 53.545, -188.556]
  MoveL 1064 to (-890, 1050, -0.5) mm, rotated rx 180 ry 0 rz 90 deg; joints [11.387, -80.812, 137.134, 193.605, 57.071, -187.495]
  MoveL 1065 to (-890, 1050, 50) mm, rotated rx -180 ry 0 rz 90 deg; joints [11.387, -84, 136.691, 194.209, 53.545, -188.556]
  MoveL 1066 to (-890, 1100, 50) mm, rotated rx -180 ry 0 rz 90 deg; joints [11.894, -86.184, 139.185, 194.774, 53.922, -188.828]
  MoveL 1067 to (-890, 1100, -0.5) mm, rotated rx 180 ry 0 rz 90 deg; joints [11.894, -82.807, 139.652, 194.122, 57.644, -187.668]
  MoveL 1068 to (-890, 1100, 50) mm, rotated rx -180 ry 0 rz 90 deg; joints [11.894, -86.184, 139.185, 194.774, 53.922, -188.828]
  MoveL 1069 to (-890, 1150, 50) mm, rotated rx 180 ry 0 rz 90 deg; joints [12.447, -88.469, 141.648, 195.415, 54.181, -189.167]
  MoveL 1070 to (-890, 1150, -0.5) mm, rotated rx -180 ry 0 rz 90 deg; joints [12.447, -84.884, 142.143, 194.704, 58.12, -187.891]
  MoveL 1071 to (-890, 1150, 50) mm, rotated rx 180 ry 0 rz 90 deg; joints [12.447, -88.469, 141.648, 195.415, 54.181, -189.167]
  MoveL 1072 to (-890, 1200, 50) mm, rotated rx -180 ry 0 rz 90 deg; joints [13.054, -90.879, 144.081, 196.148, 54.302, -189.59]
  MoveL 1073 to (-890, 1200, -0.5) mm, rotated rx 180 ry 0 rz 90 deg; joints [13.054, -87.061, 144.607, 195.364, 58.483, -188.174]
  MoveL 1074 to (-890, 1200, 50) mm, rotated rx -180 ry 0 rz 90 deg; joints [13.054, -90.879, 144.081, 196.148, 54.302, -189.59]
  MoveL 1075 to (-890, 1250, 50) mm, rotated rx 180 ry 0 rz 90 deg; joints [13.721, -93.443, 146.484, 196.991, 54.261, -190.119]
  MoveL 1076 to (-890, 1250, -0.5) mm, rotated rx 180 ry 0 rz 90 deg; joints [13.721, -89.364, 147.045, 196.115, 58.71, -188.534]
  MoveL 1077 to (-890, 1250, 50) mm, rotated rx 180 ry 0 rz 90 deg; joints [13.721, -93.443, 146.484, 196.991, 54.261, -190.119]
  MoveL 1078 to (-890, 1300, 50) mm, rotated rx -180 ry 0 rz 90 deg; joints [14.459, -96.198, 148.853, 197.97, 54.028, -190.786]
  MoveL 1079 to (-890, 1300, -0.5) mm, rotated rx -180 ry 0 rz 90 deg; joints [14.459, -91.824, 149.457, 196.976, 58.776, -188.992]
  MoveL 1080 to (-890, 1300, 50) mm, rotated rx -180 ry 0 rz 90 deg; joints [14.459, -96.198, 148.853, 197.97, 54.028, -190.786]
  MoveL 1081 to (-890, 1350, 50) mm, rotated rx -180 ry 0 rz 90 deg; joints [15.278, -99.19, 151.188, 199.119, 53.564, -191.634]
  MoveL 1082 to (-890, 1350, -0.5) mm, rotated rx 180 ry 0 rz 90 deg; joints [15.278, -94.484, 151.841, 197.973, 58.646, -189.581]
  MoveL 1083 to (-890, 1350, 50) mm, rotated rx -180 ry 0 rz 90 deg; joints [15.278, -99.19, 151.188, 199.119, 53.564, -191.634]
  MoveL 1084 to (-890, 1400, 50) mm, rotated rx -180 ry 0 rz 90 deg; joints [16.194, -102.482, 153.485, 200.489, 52.821, -192.724]
  MoveL 1085 to (-890, 1400, -0.5) mm, rotated rx 180 ry 0 rz 90 deg; joints [16.194, -97.401, 154.196, 199.141, 58.271, -190.344]
  MoveL 1086 to (-890, 1400, 50) mm, rotated rx -180 ry 0 rz 90 deg; joints [16.194, -102.482, 153.485, 200.489, 52.821, -192.724]
  MoveL 1087 to (-890, 1450, 50) mm, rotated rx -180 ry 0 rz 110 deg; joints [23.693, -102.084, 153.222, 230.82, 63.02, -209.102]
  MoveL 1088 to (-890, 1450, -0.5) mm, rotated rx -180 ry 0 rz 110 deg; joints [23.693, -97.049, 153.926, 228.762, 66.728, -204.262]
  MoveL 1089 to (-890, 1450, 50) mm, rotated rx -180 ry 0 rz 110 deg; joints [23.693, -102.084, 153.222, 230.82, 63.02, -209.102]
  MoveL 1090 to (-960, 50, 50) mm, rotated rx 180 ry 0 rz 90 deg; joints [7.973, -45.453, 76.566, 195.165, 32.019, -192.942]
  MoveL 1091 to (-960, 50, -0.5) mm, rotated rx -180 ry 0 rz 90 deg; joints [7.973, -44.021, 76.864, 194.48, 33.691, -192.127]
  MoveL 1092 to (-960, 50, 50) mm, rotated rx 180 ry 0 rz 90 deg; joints [7.973, -45.453, 76.566, 195.165, 32.019, -192.942]
  MoveL 1093 to (-960, 100, 50) mm, rotated rx -180 ry 0 rz 90 deg; joints [8.161, -47.53, 80.293, 194.842, 33.654, -192.439]
  MoveL 1094 to (-960, 100, -0.5) mm, rotated rx 180 ry 0 rz 90 deg; joints [8.161, -46.052, 80.587, 194.196, 35.369, -191.655]
  MoveL 1095 to (-960, 100, 50) mm, rotated rx -180 ry 0 rz 90 deg; joints [8.161, -47.53, 80.293, 194.842, 33.654, -192.439]
  MoveL 1096 to (-960, 150, 50) mm, rotated rx -180 ry 0 rz 90 deg; joints [8.358, -49.548, 83.882, 194.6, 35.216, -192.014]
  MoveL 1097 to (-960, 150, -0.5) mm, rotated rx 180 ry 0 rz 90 deg; joints [8.358, -48.023, 84.175, 193.984, 36.977, -191.252]
  MoveL 1098 to (-960, 150, 50) mm, rotated rx -180 ry 0 rz 90 deg; joints [8.358, -49.548, 83.882, 194.6, 35.216, -192.014]
  MoveL 1099 to (-960, 200, 50) mm, rotated rx 180 ry 0 rz 90 deg; joints [8.565, -51.516, 87.353, 194.426, 36.712, -191.652]
  MoveL 1100 to (-960, 200, -0.5) mm, rotated rx -180 ry 0 rz 90 deg; joints [8.565, -49.942, 87.644, 193.834, 38.521, -190.906]
  MoveL 1101 to (-960, 200, 50) mm, rotated rx 180 ry 0 rz 90 deg; joints [8.565, -51.516, 87.353, 194.426, 36.712, -191.652]
  MoveL 1102 to (-960, 250, 50) mm, rotated rx 180 ry 0 rz 90 deg; joints [8.782, -53.444, 90.717, 194.31, 38.147, -191.343]
  MoveL 1103 to (-960, 250, -0.5) mm, rotated rx -180 ry 0 rz 90 deg; joints [8.782, -51.818, 91.009, 193.738, 40.007, -190.606]
  MoveL 1104 to (-960, 250, 50) mm, rotated rx 180 ry 0 rz 90 deg; joints [8.782, -53.444, 90.717, 194.31, 38.147, -191.343]
  MoveL 1105 to (-960, 300, 50) mm, rotated rx 180 ry 0 rz 90 deg; joints [9.01, -55.337, 93.986, 194.245, 39.525, -191.08]
  MoveL 1106 to (-960, 300, -0.5) mm, rotated rx 180 ry 0 rz 90 deg; joints [9.01, -53.657, 94.279, 193.687, 41.44, -190.347]
  MoveL 1107 to (-960, 300, 50) mm, rotated rx 180 ry 0 rz 90 deg; joints [9.01, -55.337, 93.986, 194.245, 39.525, -191.08]
  MoveL 1108 to (-960, 350, 50) mm, rotated rx -180 ry 0 rz 90 deg; joints [9.25, -57.202, 97.171, 194.227, 40.85, -190.857]
  MoveL 1109 to (-960, 350, -0.5) mm, rotated rx 180 ry 0 rz 90 deg; joints [9.25, -55.465, 97.466, 193.679, 42.822, -190.122]
  MoveL 1110 to (-960, 350, 50) mm, rotated rx -180 ry 0 rz 90 deg; joints [9.25, -57.202, 97.171, 194.227, 40.85, -190.857]
  MoveL 1111 to (-960, 400, 50) mm, rotated rx 180 ry 0 rz 90 deg; joints [9.504, -59.044, 100.278, 194.251, 42.123, -190.668]
  MoveL 1112 to (-960, 400, -0.5) mm, rotated rx 180 ry 0 rz 90 deg; joints [9.504, -57.247, 100.577, 193.711, 44.157, -189.928]
  MoveL 1113 to (-960, 400, 50) mm, rotated rx 180 ry 0 rz 90 deg; joints [9.504, -59.044, 100.278, 194.251, 42.123, -190.668]
  MoveL 1114 to (-960, 450, 50) mm, rotated rx -180 ry 0 rz 90 deg; joints [9.771, -60.869, 103.316, 194.315, 43.348, -190.512]
  MoveL 1115 to (-960, 450, -0.5) mm, rotated rx 180 ry 0 rz 90 deg; joints [9.771, -59.008, 103.618, 193.778, 45.447, -189.762]
  MoveL 1116 to (-960, 450, 50) mm, rotated rx -180 ry 0 rz 90 deg; joints [9.771, -60.869, 103.316, 194.315, 43.348, -190.512]
  MoveL 1117 to (-960, 500, 50) mm, rotated rx 180 ry 0 rz 90 deg; joints [10.054, -62.682, 106.289, 194.417, 44.524, -190.386]
  MoveL 1118 to (-960, 500, -0.5) mm, rotated rx 180 ry 0 rz 90 deg; joints [10.054, -60.753, 106.597, 193.882, 46.692, -189.621]
  MoveL 1119 to (-960, 500, 50) mm, rotated rx 180 ry 0 rz 90 deg; joints [10.054, -62.682, 106.289, 194.417, 44.524, -190.386]
  MoveL 1120 to (-960, 550, 50) mm, rotated rx 180 ry 0 rz 90 deg; joints [10.354, -64.487, 109.204, 194.556, 45.652, -190.288]
  MoveL 1121 to (-960, 550, -0.5) mm, rotated rx 180 ry 0 rz 90 deg; joints [10.354, -62.485, 109.517, 194.019, 47.895, -189.504]
  MoveL 1122 to (-960, 550, 50) mm, rotated rx 180 ry 0 rz 90 deg; joints [10.354, -64.487, 109.204, 194.556, 45.652, -190.288]
  MoveL 1123 to (-960, 600, 50) mm, rotated rx -180 ry 0 rz 90 deg; joints [10.672, -66.29, 112.065, 194.733, 46.732, -190.217]
  MoveL 1124 to (-960, 600, -0.5) mm, rotated rx -180 ry 0 rz 90 deg; joints [10.672, -64.21, 112.384, 194.192, 49.055, -189.41]
  MoveL 1125 to (-960, 600, 50) mm, rotated rx -180 ry 0 rz 90 deg; joints [10.672, -66.29, 112.065, 194.733, 46.732, -190.217]
  MoveL 1126 to (-960, 650, 50) mm, rotated rx -180 ry 0 rz 90 deg; joints [11.01, -68.094, 114.875, 194.948, 47.764, -190.174]
  MoveL 1127 to (-960, 650, -0.5) mm, rotated rx -180 ry 0 rz 90 deg; joints [11.01, -65.931, 115.202, 194.399, 50.173, -189.338]
  MoveL 1128 to (-960, 650, 50) mm, rotated rx -180 ry 0 rz 90 deg; joints [11.01, -68.094, 114.875, 194.948, 47.764, -190.174]
  MoveL 1129 to (-960, 700, 50) mm, rotated rx -180 ry 0 rz 90 deg; joints [11.369, -69.906, 117.639, 195.201, 48.747, -190.158]
  MoveL 1130 to (-960, 700, -0.5) mm, rotated rx -180 ry 0 rz 90 deg; joints [11.369, -67.654, 117.975, 194.642, 51.248, -189.288]
  MoveL 1131 to (-960, 700, 50) mm, rotated rx -180 ry 0 rz 90 deg; joints [11.369, -69.906, 117.639, 195.201, 48.747, -190.158]
  MoveL 1132 to (-960, 750, 50) mm, rotated rx -180 ry 0 rz 90 deg; joints [11.752, -71.73, 120.359, 195.495, 49.678, -190.17]
  MoveL 1133 to (-960, 750, -0.5) mm, rotated rx -180 ry 0 rz 90 deg; joints [11.752, -69.381, 120.704, 194.922, 52.278, -189.26]
  MoveL 1134 to (-960, 750, 50) mm, rotated rx -180 ry 0 rz 90 deg; joints [11.752, -71.73, 120.359, 195.495, 49.678, -190.17]
  MoveL 1135 to (-960, 800, 50) mm, rotated rx -180 ry 0 rz 90 deg; joints [12.162, -73.572, 123.037, 195.832, 50.556, -190.213]
  MoveL 1136 to (-960, 800, -0.5) mm, rotated rx -180 ry 0 rz 90 deg; joints [12.162, -71.12, 123.394, 195.242, 53.263, -189.257]
  MoveL 1137 to (-960, 800, 50) mm, rotated rx -180 ry 0 rz 90 deg; joints [12.162, -73.572, 123.037, 195.832, 50.556, -190.213]
  MoveL 1138 to (-960, 850, 50) mm, rotated rx 180 ry 0 rz 90 deg; joints [12.601, -75.44, 125.677, 196.215, 51.376, -190.289]
  MoveL 1139 to (-960, 850, -0.5) mm, rotated rx 180 ry 0 rz 90 deg; joints [12.601, -72.874, 126.046, 195.604, 54.199, -189.278]
  MoveL 1140 to (-960, 850, 50) mm, rotated rx 180 ry 0 rz 90 deg; joints [12.601, -75.44, 125.677, 196.215, 51.376, -190.289]
  MoveL 1141 to (-960, 900, 50) mm, rotated rx 180 ry 0 rz 90 deg; joints [13.072, -77.339, 128.28, 196.648, 52.136, -190.4]
  MoveL 1142 to (-960, 900, -0.5) mm, rotated rx 180 ry 0 rz 90 deg; joints [13.072, -74.65, 128.663, 196.012, 55.084, -189.328]
  MoveL 1143 to (-960, 900, 50) mm, rotated rx 180 ry 0 rz 90 deg; joints [13.072, -77.339, 128.28, 196.648, 52.136, -190.4]
  MoveL 1144 to (-960, 950, 50) mm, rotated rx -180 ry 0 rz 90 deg; joints [13.579, -79.278, 130.847, 197.137, 52.83, -190.553]
  MoveL 1145 to (-960, 950, -0.5) mm, rotated rx 180 ry 0 rz 90 deg; joints [13.579, -76.454, 131.246, 196.469, 55.914, -189.407]
  MoveL 1146 to (-960, 950, 50) mm, rotated rx -180 ry 0 rz 90 deg; joints [13.579, -79.278, 130.847, 197.137, 52.83, -190.553]
  MoveL 1147 to (-960, 1000, 50) mm, rotated rx 180 ry 0 rz 90 deg; joints [14.127, -81.266, 133.38, 197.687, 53.451, -190.753]
  MoveL 1148 to (-960, 1000, -0.5) mm, rotated rx 180 ry 0 rz 90 deg; joints [14.127, -78.295, 133.797, 196.982, 56.684, -189.522]
  MoveL 1149 to (-960, 1000, 50) mm, rotated rx 180 ry 0 rz 90 deg; joints [14.127, -81.266, 133.38, 197.687, 53.451, -190.753]
  MoveL 1150 to (-960, 1050, 50) mm, rotated rx -180 ry 0 rz 90 deg; joints [14.719, -83.315, 135.88, 198.306, 53.991, -191.007]
  MoveL 1151 to (-960, 1050, -0.5) mm, rotated rx -180 ry 0 rz 90 deg; joints [14.719, -80.182, 136.316, 197.556, 57.387, -189.677]
  MoveL 1152 to (-960, 1050, 50) mm, rotated rx -180 ry 0 rz 90 deg; joints [14.719, -83.315, 135.88, 198.306, 53.991, -191.007]
  MoveL 1153 to (-960, 1100, 50) mm, rotated rx 180 ry 0 rz 90 deg; joints [15.362, -85.437, 138.347, 199.004, 54.442, -191.325]
  MoveL 1154 to (-960, 1100, -0.5) mm, rotated rx -180 ry 0 rz 90 deg; joints [15.362, -82.126, 138.806, 198.199, 58.015, -189.879]
  MoveL 1155 to (-960, 1100, 50) mm, rotated rx 180 ry 0 rz 90 deg; joints [15.362, -85.437, 138.347, 199.004, 54.442, -191.325]
  MoveL 1156 to (-960, 1150, 50) mm, rotated rx -180 ry 0 rz 90 deg; joints [16.062, -87.649, 140.782, 199.792, 54.792, -191.722]
  MoveL 1157 to (-960, 1150, -0.5) mm, rotated rx -180 ry 0 rz 90 deg; joints [16.062, -84.14, 141.266, 198.922, 58.56, -190.138]
  MoveL 1158 to (-960, 1150, 50) mm, rotated rx -180 ry 0 rz 90 deg; joints [16.062, -87.649, 140.782, 199.792, 54.792, -191.722]
  MoveL 1159 to (-960, 1200, 50) mm, rotated rx -180 ry 0 rz 90 deg; joints [16.826, -89.97, 143.183, 200.687, 55.027, -192.213]
  MoveL 1160 to (-960, 1200, -0.5) mm, rotated rx 180 ry 0 rz 90 deg; joints [16.826, -86.241, 143.697, 199.736, 59.008, -190.466]
  MoveL 1161 to (-960, 1200, 50) mm, rotated rx -180 ry 0 rz 90 deg; joints [16.826, -89.97, 143.183, 200.687, 55.027, -192.213]
  MoveL 1162 to (-960, 1250, 50) mm, rotated rx -180 ry 0 rz 90 deg; joints [17.665, -92.423, 145.551, 201.708, 55.128, -192.823]
  MoveL 1163 to (-960, 1250, -0.5) mm, rotated rx 180 ry 0 rz 90 deg; joints [17.665, -88.449, 146.098, 200.656, 59.344, -190.88]
  MoveL 1164 to (-960, 1250, 50) mm, rotated rx -180 ry 0 rz 90 deg; joints [17.665, -92.423, 145.551, 201.708, 55.128, -192.823]
  MoveL 1165 to (-960, 1300, 50) mm, rotated rx 180 ry 0 rz 90 deg; joints [18.589, -95.039, 147.883, 202.879, 55.077, -193.581]
  MoveL 1166 to (-960, 1300, -0.5) mm, rotated rx -180 ry 0 rz 90 deg; joints [18.589, -90.791, 148.469, 201.702, 59.55, -191.403]
  MoveL 1167 to (-960, 1300, 50) mm, rotated rx 180 ry 0 rz 90 deg; joints [18.589, -95.039, 147.883, 202.879, 55.077, -193.581]
  MoveL 1168 to (-960, 1350, 50) mm, rotated rx -180 ry 0 rz 90 deg; joints [19.611, -97.855, 150.177, 204.236, 54.846, -194.531]
  MoveL 1169 to (-960, 1350, -0.5) mm, rotated rx 180 ry 0 rz 90 deg; joints [19.611, -93.299, 150.808, 202.9, 59.602, -192.065]
  MoveL 1170 to (-960, 1350, 50) mm, rotated rx -180 ry 0 rz 90 deg; joints [19.611, -97.855, 150.177, 204.236, 54.846, -194.531]
  MoveL 1171 to (-960, 1400, 50) mm, rotated rx -180 ry 0 rz 90 deg; joints [20.746, -100.92, 152.43, 205.824, 54.407, -195.731]
  MoveL 1172 to (-960, 1400, -0.5) mm, rotated rx -180 ry 0 rz 90 deg; joints [20.746, -96.017, 153.113, 204.283, 59.468, -192.909]
  MoveL 1173 to (-960, 1400, 50) mm, rotated rx -180 ry 0 rz 90 deg; joints [20.746, -100.92, 152.43, 205.824, 54.407, -195.731]
  MoveL 1174 to (-960, 1450, 50) mm, rotated rx 180 ry 0 rz 90 deg; joints [22.014, -104.295, 154.636, 207.708, 53.723, -197.262]
  MoveL 1175 to (-960, 1450, -0.5) mm, rotated rx -180 ry 0 rz 110 deg; joints [27.964, -95.187, 152.434, 232.83, 68.76, -205.538]
  MoveL 1176 to (-960, 1450, 50) mm, rotated rx 180 ry 0 rz 90 deg; joints [22.014, -104.295, 154.636, 207.708, 53.723, -197.262]
  MoveL 1177 to (-1030, 50, 50) mm, rotated rx -180 ry 0 rz 90 deg; joints [9.8, -44.991, 75.733, 198.671, 32.12, -195.971]
  MoveL 1178 to (-1030, 50, -0.5) mm, rotated rx 180 ry 0 rz 90 deg; joints [9.8, -43.568, 76.031, 197.839, 33.754, -194.98]
  MoveL 1179 to (-1030, 50, 50) mm, rotated rx -180 ry 0 rz 90 deg; joints [9.8, -44.991, 75.733, 198.671, 32.12, -195.971]
  MoveL 1180 to (-1030, 100, 50) mm, rotated rx 180 ry 0 rz 90 deg; joints [10.03, -47.071, 79.472, 198.266, 33.756, -195.346]
  MoveL 1181 to (-1030, 100, -0.5) mm, rotated rx 180 ry 0 rz 90 deg; joints [10.03, -45.603, 79.767, 197.482, 35.433, -194.393]
  MoveL 1182 to (-1030, 100, 50) mm, rotated rx 180 ry 0 rz 90 deg; joints [10.03, -47.071, 79.472, 198.266, 33.756, -195.346]
  MoveL 1183 to (-1030, 150, 50) mm, rotated rx 180 ry 0 rz 90 deg; joints [10.27, -49.09, 83.071, 197.962, 35.32, -194.816]
  MoveL 1184 to (-1030, 150, -0.5) mm, rotated rx -180 ry 0 rz 90 deg; joints [10.27, -47.576, 83.364, 197.216, 37.042, -193.892]
  MoveL 1185 to (-1030, 150, 50) mm, rotated rx 180 ry 0 rz 90 deg; joints [10.27, -49.09, 83.071, 197.962, 35.32, -194.816]
  MoveL 1186 to (-1030, 200, 50) mm, rotated rx 180 ry 0 rz 90 deg; joints [10.522, -51.058, 86.548, 197.741, 36.82, -194.366]
  MoveL 1187 to (-1030, 200, -0.5) mm, rotated rx 180 ry 0 rz 90 deg; joints [10.522, -49.496, 86.84, 197.025, 38.589, -193.46]
  MoveL 1188 to (-1030, 200, 50) mm, rotated rx 180 ry 0 rz 90 deg; joints [10.522, -51.058, 86.548, 197.741, 36.82, -194.366]
  MoveL 1189 to (-1030, 250, 50) mm, rotated rx -180 ry 0 rz 90 deg; joints [10.787, -52.983, 89.916, 197.593, 38.259, -193.981]
  MoveL 1190 to (-1030, 250, -0.5) mm, rotated rx -180 ry 0 rz 90 deg; joints [10.787, -51.37, 90.208, 196.899, 40.078, -193.087]
  MoveL 1191 to (-1030, 250, 50) mm, rotated rx -180 ry 0 rz 90 deg; joints [10.787, -52.983, 89.916, 197.593, 38.259, -193.981]
  MoveL 1192 to (-1030, 300, 50) mm, rotated rx 180 ry 0 rz 90 deg; joints [11.065, -54.872, 93.187, 197.507, 39.643, -193.652]
  MoveL 1193 to (-1030, 300, -0.5) mm, rotated rx 180 ry 0 rz 90 deg; joints [11.065, -53.206, 93.479, 196.832, 41.515, -192.763]
  MoveL 1194 to (-1030, 300, 50) mm, rotated rx 180 ry 0 rz 90 deg; joints [11.065, -54.872, 93.187, 197.507, 39.643, -193.652]
  MoveL 1195 to (-1030, 350, 50) mm, rotated rx 180 ry 0 rz 90 deg; joints [11.358, -56.731, 96.37, 197.477, 40.975, -193.372]
  MoveL 1196 to (-1030, 350, -0.5) mm, rotated rx -180 ry 0 rz 90 deg; joints [11.358, -55.009, 96.665, 196.815, 42.902, -192.483]
  MoveL 1197 to (-1030, 350, 50) mm, rotated rx 180 ry 0 rz 90 deg; joints [11.358, -56.731, 96.37, 197.477, 40.975, -193.372]
  MoveL 1198 to (-1030, 400, 50) mm, rotated rx -180 ry 0 rz 90 deg; joints [11.666, -58.565, 99.475, 197.5, 42.257, -193.135]
  MoveL 1199 to (-1030, 400, -0.5) mm, rotated rx 180 ry 0 rz 90 deg; joints [11.666, -56.784, 99.772, 196.847, 44.243, -192.24]
  MoveL 1200 to (-1030, 400, 50) mm, rotated rx -180 ry 0 rz 90 deg; joints [11.666, -58.565, 99.475, 197.5, 42.257, -193.135]
  MoveL 1201 to (-1030, 450, 50) mm, rotated rx -180 ry 0 rz 90 deg; joints [11.991, -60.381, 102.508, 197.57, 43.491, -192.938]
  MoveL 1202 to (-1030, 450, -0.5) mm, rotated rx 180 ry 0 rz 90 deg; joints [11.991, -58.537, 102.809, 196.924, 45.54, -192.031]
  MoveL 1203 to (-1030, 450, 50) mm, rotated rx -180 ry 0 rz 90 deg; joints [11.991, -60.381, 102.508, 197.57, 43.491, -192.938]
  MoveL 1204 to (-1030, 500, 50) mm, rotated rx 180 ry 0 rz 90 deg; joints [12.335, -62.182, 105.475, 197.688, 44.678, -192.776]
  MoveL 1205 to (-1030, 500, -0.5) mm, rotated rx -180 ry 0 rz 90 deg; joints [12.335, -60.272, 105.78, 197.043, 46.793, -191.853]
  MoveL 1206 to (-1030, 500, 50) mm, rotated rx 180 ry 0 rz 90 deg; joints [12.335, -62.182, 105.475, 197.688, 44.678, -192.776]
  MoveL 1207 to (-1030, 550, 50) mm, rotated rx 180 ry 0 rz 90 deg; joints [12.699, -63.974, 108.381, 197.85, 45.82, -192.649]
  MoveL 1208 to (-1030, 550, -0.5) mm, rotated rx -180 ry 0 rz 90 deg; joints [12.699, -61.993, 108.692, 197.204, 48.006, -191.704]
  MoveL 1209 to (-1030, 550, 50) mm, rotated rx 180 ry 0 rz 90 deg; joints [12.699, -63.974, 108.381, 197.85, 45.82, -192.649]
  MoveL 1210 to (-1030, 600, 50) mm, rotated rx -180 ry 0 rz 90 deg; joints [13.084, -65.761, 111.231, 198.057, 46.916, -192.554]
  MoveL 1211 to (-1030, 600, -0.5) mm, rotated rx 180 ry 0 rz 90 deg; joints [13.084, -63.705, 111.549, 197.407, 49.177, -191.582]
  MoveL 1212 to (-1030, 600, 50) mm, rotated rx -180 ry 0 rz 90 deg; joints [13.084, -65.761, 111.231, 198.057, 46.916, -192.554]
  MoveL 1213 to (-1030, 650, 50) mm, rotated rx 180 ry 0 rz 90 deg; joints [13.493, -67.547, 114.03, 198.309, 47.966, -192.492]
  MoveL 1214 to (-1030, 650, -0.5) mm, rotated rx -180 ry 0 rz 90 deg; joints [13.493, -65.411, 114.355, 197.651, 50.307, -191.488]
  MoveL 1215 to (-1030, 650, 50) mm, rotated rx 180 ry 0 rz 90 deg; joints [13.493, -67.547, 114.03, 198.309, 47.966, -192.492]
  MoveL 1216 to (-1030, 700, 50) mm, rotated rx 180 ry 0 rz 90 deg; joints [13.928, -69.338, 116.779, 198.607, 48.969, -192.463]
  MoveL 1217 to (-1030, 700, -0.5) mm, rotated rx 180 ry 0 rz 90 deg; joints [13.928, -67.115, 117.113, 197.939, 51.397, -191.419]
  MoveL 1218 to (-1030, 700, 50) mm, rotated rx 180 ry 0 rz 90 deg; joints [13.928, -69.338, 116.779, 198.607, 48.969, -192.463]
  MoveL 1219 to (-1030, 750, 50) mm, rotated rx 180 ry 0 rz 90 deg; joints [14.391, -71.138, 119.484, 198.953, 49.925, -192.467]
  MoveL 1220 to (-1030, 750, -0.5) mm, rotated rx -180 ry 0 rz 90 deg; joints [14.391, -68.822, 119.826, 198.271, 52.445, -191.378]
  MoveL 1221 to (-1030, 750, 50) mm, rotated rx 180 ry 0 rz 90 deg; joints [14.391, -71.138, 119.484, 198.953, 49.925, -192.467]
  MoveL 1222 to (-1030, 800, 50) mm, rotated rx -180 ry 0 rz 90 deg; joints [14.885, -72.953, 122.145, 199.35, 50.832, -192.506]
  MoveL 1223 to (-1030, 800, -0.5) mm, rotated rx 180 ry 0 rz 90 deg; joints [14.885, -70.536, 122.497, 198.649, 53.451, -191.364]
  MoveL 1224 to (-1030, 800, 50) mm, rotated rx -180 ry 0 rz 90 deg; joints [14.885, -72.953, 122.145, 199.35, 50.832, -192.506]
  MoveL 1225 to (-1030, 850, 50) mm, rotated rx -180 ry 0 rz 90 deg; joints [15.414, -74.788, 124.765, 199.801, 51.686, -192.583]
  MoveL 1226 to (-1030, 850, -0.5) mm, rotated rx 180 ry 0 rz 90 deg; joints [15.414, -72.263, 125.129, 199.077, 54.412, -191.379]
  MoveL 1227 to (-1030, 850, 50) mm, rotated rx -180 ry 0 rz 90 deg; joints [15.414, -74.788, 124.765, 199.801, 51.686, -192.583]
  MoveL 1228 to (-1030, 900, 50) mm, rotated rx 180 ry 0 rz 90 deg; joints [15.981, -76.65, 127.346, 200.309, 52.486, -192.701]
  MoveL 1229 to (-1030, 900, -0.5) mm, rotated rx 180 ry 0 rz 90 deg; joints [15.981, -74.007, 127.724, 199.558, 55.326, -191.426]
  MoveL 1230 to (-1030, 900, 50) mm, rotated rx 180 ry 0 rz 90 deg; joints [15.981, -76.65, 127.346, 200.309, 52.486, -192.701]
  MoveL 1231 to (-1030, 950, 50) mm, rotated rx 180 ry 0 rz 90 deg; joints [16.589, -78.546, 129.889, 200.881, 53.227, -192.865]
  MoveL 1232 to (-1030, 950, -0.5) mm, rotated rx -180 ry 0 rz 90 deg; joints [16.589, -75.774, 130.282, 200.097, 56.191, -191.508]
  MoveL 1233 to (-1030, 950, 50) mm, rotated rx 180 ry 0 rz 90 deg; joints [16.589, -78.546, 129.889, 200.881, 53.227, -192.865]
  MoveL 1234 to (-1030, 1000, 50) mm, rotated rx -180 ry 0 rz 90 deg; joints [17.244, -80.483, 132.396, 201.523, 53.904, -193.08]
  MoveL 1235 to (-1030, 1000, -0.5) mm, rotated rx -180 ry 0 rz 90 deg; joints [17.244, -77.572, 132.805, 200.7, 57.002, -191.628]
  MoveL 1236 to (-1030, 1000, 50) mm, rotated rx -180 ry 0 rz 90 deg; joints [17.244, -80.483, 132.396, 201.523, 53.904, -193.08]
  MoveL 1237 to (-1030, 1050, 50) mm, rotated rx 180 ry 0 rz 90 deg; joints [17.952, -82.473, 134.867, 202.243, 54.513, -193.355]
  MoveL 1238 to (-1030, 1050, -0.5) mm, rotated rx 180 ry 0 rz 90 deg; joints [17.952, -79.408, 135.294, 201.372, 57.756, -191.793]
  MoveL 1239 to (-1030, 1050, 50) mm, rotated rx 180 ry 0 rz 90 deg; joints [17.952, -82.473, 134.867, 202.243, 54.513, -193.355]
  MoveL 1240 to (-1030, 1100, 50) mm, rotated rx 180 ry 0 rz 90 deg; joints [18.718, -84.524, 137.302, 203.05, 55.046, -193.7]
  MoveL 1241 to (-1030, 1100, -0.5) mm, rotated rx -180 ry 0 rz 90 deg; joints [18.718, -81.292, 137.751, 202.123, 58.445, -192.01]
  MoveL 1242 to (-1030, 1100, 50) mm, rotated rx 180 ry 0 rz 90 deg; joints [18.718, -84.524, 137.302, 203.05, 55.046, -193.7]
  MoveL 1243 to (-1030, 1150, 50) mm, rotated rx -180 ry 0 rz 90 deg; joints [19.549, -86.652, 139.702, 203.957, 55.496, -194.128]
  MoveL 1244 to (-1030, 1150, -0.5) mm, rotated rx -180 ry 0 rz 90 deg; joints [19.549, -83.234, 140.174, 202.961, 59.065, -192.287]
  MoveL 1245 to (-1030, 1150, 50) mm, rotated rx -180 ry 0 rz 90 deg; joints [19.549, -86.652, 139.702, 203.957, 55.496, -194.128]
  MoveL 1246 to (-1030, 1200, 50) mm, rotated rx 180 ry 0 rz 90 deg; joints [20.455, -88.87, 142.065, 204.978, 55.853, -194.654]
  MoveL 1247 to (-1030, 1200, -0.5) mm, rotated rx -180 ry 0 rz 90 deg; joints [20.455, -85.248, 142.565, 203.9, 59.606, -192.637]
  MoveL 1248 to (-1030, 1200, 50) mm, rotated rx 180 ry 0 rz 90 deg; joints [20.455, -88.87, 142.065, 204.978, 55.853, -194.654]
  MoveL 1249 to (-1030, 1250, 50) mm, rotated rx -180 ry 0 rz 90 deg; joints [21.444, -91.199, 144.392, 206.131, 56.106, -195.3]
  MoveL 1250 to (-1030, 1250, -0.5) mm, rotated rx 180 ry 0 rz 90 deg; joints [21.444, -87.349, 144.922, 204.955, 60.059, -193.076]
  MoveL 1251 to (-1030, 1250, 50) mm, rotated rx -180 ry 0 rz 90 deg; joints [21.444, -91.199, 144.392, 206.131, 56.106, -195.3]
  MoveL 1252 to (-1030, 1300, 50) mm, rotated rx -180 ry 0 rz 90 deg; joints [22.529, -93.661, 146.679, 207.441, 56.244, -196.095]
  MoveL 1253 to (-1030, 1300, -0.5) mm, rotated rx 180 ry 0 rz 90 deg; joints [22.529, -89.559, 147.244, 206.142, 60.411, -193.623]
  MoveL 1254 to (-1030, 1300, 50) mm, rotated rx -180 ry 0 rz 90 deg; joints [22.529, -93.661, 146.679, 207.441, 56.244, -196.095]
  MoveL 1255 to (-1030, 1350, 50) mm, rotated rx -180 ry 0 rz 90 deg; joints [23.722, -96.284, 148.925, 208.936, 56.252, -197.074]
  MoveL 1256 to (-1030, 1350, -0.5) mm, rotated rx 180 ry 0 rz 90 deg; joints [23.722, -91.901, 149.53, 207.487, 60.649, -194.307]
  MoveL 1257 to (-1030, 1350, 50) mm, rotated rx -180 ry 0 rz 90 deg; joints [23.722, -96.284, 148.925, 208.936, 56.252, -197.074]
  MoveL 1258 to (-1030, 1400, 50) mm, rotated rx -180 ry 0 rz 90 deg; joints [25.041, -99.104, 151.125, 210.654, 56.115, -198.286]
  MoveL 1259 to (-1030, 1400, -0.5) mm, rotated rx 180 ry 0 rz 90 deg; joints [25.041, -94.408, 151.777, 209.019, 60.755, -195.164]
  MoveL 1260 to (-1030, 1400, 50) mm, rotated rx -180 ry 0 rz 90 deg; joints [25.041, -99.104, 151.125, 210.654, 56.115, -198.286]
  MoveL 1261 to (-1100, 50, 50) mm, rotated rx 180 ry 0 rz 90 deg; joints [11.608, -44.43, 74.72, 202.16, 32.239, -199.008]
  MoveL 1262 to (-1100, 50, -0.5) mm, rotated rx 180 ry 0 rz 90 deg; joints [11.608, -43.019, 75.019, 201.188, 33.829, -197.849]
  MoveL 1263 to (-1100, 50, 50) mm, rotated rx 180 ry 0 rz 90 deg; joints [11.608, -44.43, 74.72, 202.16, 32.239, -199.008]
  MoveL 1264 to (-1100, 100, 50) mm, rotated rx 180 ry 0 rz 90 deg; joints [11.878, -46.515, 78.476, 201.67, 33.876, -198.257]
  MoveL 1265 to (-1100, 100, -0.5) mm, rotated rx 180 ry 0 rz 90 deg; joints [11.878, -45.06, 78.772, 200.754, 35.509, -197.144]
  MoveL 1266 to (-1100, 100, 50) mm, rotated rx 180 ry 0 rz 90 deg; joints [11.878, -46.515, 78.476, 201.67, 33.876, -198.257]
  MoveL 1267 to (-1100, 150, 50) mm, rotated rx 180 ry 0 rz 90 deg; joints [12.16, -48.537, 82.088, 201.299, 35.443, -197.621]
  MoveL 1268 to (-1100, 150, -0.5) mm, rotated rx -180 ry 0 rz 90 deg; joints [12.16, -47.036, 82.381, 200.429, 37.12, -196.541]
  MoveL 1269 to (-1100, 150, 50) mm, rotated rx 180 ry 0 rz 90 deg; joints [12.16, -48.537, 82.088, 201.299, 35.443, -197.621]
  MoveL 1270 to (-1100, 200, 50) mm, rotated rx -180 ry 0 rz 90 deg; joints [12.456, -50.505, 85.573, 201.029, 36.946, -197.079]
  MoveL 1271 to (-1100, 200, -0.5) mm, rotated rx 180 ry 0 rz 90 deg; joints [12.456, -48.956, 85.865, 200.194, 38.669, -196.022]
  MoveL 1272 to (-1100, 200, 50) mm, rotated rx -180 ry 0 rz 90 deg; joints [12.456, -50.505, 85.573, 201.029, 36.946, -197.079]
  MoveL 1273 to (-1100, 250, 50) mm, rotated rx -180 ry 0 rz 90 deg; joints [12.766, -52.427, 88.947, 200.843, 38.391, -196.616]
  MoveL 1274 to (-1100, 250, -0.5) mm, rotated rx 180 ry 0 rz 90 deg; joints [12.766, -50.829, 89.238, 200.036, 40.162, -195.573]
  MoveL 1275 to (-1100, 250, 50) mm, rotated rx -180 ry 0 rz 90 deg; joints [12.766, -52.427, 88.947, 200.843, 38.391, -196.616]
  MoveL 1276 to (-1100, 300, 50) mm, rotated rx -180 ry 0 rz 90 deg; joints [13.092, -54.311, 92.22, 200.732, 39.782, -196.219]
  MoveL 1277 to (-1100, 300, -0.5) mm, rotated rx 180 ry 0 rz 90 deg; joints [13.092, -52.661, 92.512, 199.947, 41.603, -195.183]
  MoveL 1278 to (-1100, 300, 50) mm, rotated rx -180 ry 0 rz 90 deg; joints [13.092, -54.311, 92.22, 200.732, 39.782, -196.219]
  MoveL 1279 to (-1100, 350, 50) mm, rotated rx 180 ry 0 rz 90 deg; joints [13.435, -56.164, 95.403, 200.688, 41.121, -195.88]
  MoveL 1280 to (-1100, 350, -0.5) mm, rotated rx 180 ry 0 rz 90 deg; joints [13.435, -54.459, 95.697, 199.919, 42.996, -194.844]
  MoveL 1281 to (-1100, 350, 50) mm, rotated rx 180 ry 0 rz 90 deg; joints [13.435, -56.164, 95.403, 200.688, 41.121, -195.88]
  MoveL 1282 to (-1100, 400, 50) mm, rotated rx 180 ry 0 rz 90 deg; joints [13.795, -57.99, 98.505, 200.704, 42.413, -195.591]
  MoveL 1283 to (-1100, 400, -0.5) mm, rotated rx 180 ry 0 rz 90 deg; joints [13.795, -56.228, 98.802, 199.947, 44.343, -194.55]
  MoveL 1284 to (-1100, 400, 50) mm, rotated rx 180 ry 0 rz 90 deg; joints [13.795, -57.99, 98.505, 200.704, 42.413, -195.591]
  MoveL 1285 to (-1100, 450, 50) mm, rotated rx 180 ry 0 rz 90 deg; joints [14.175, -59.795, 101.533, 200.777, 43.658, -195.349]
  MoveL 1286 to (-1100, 450, -0.5) mm, rotated rx -180 ry 0 rz 90 deg; joints [14.175, -57.972, 101.833, 200.028, 45.648, -194.296]
  MoveL 1287 to (-1100, 450, 50) mm, rotated rx 180 ry 0 rz 90 deg; joints [14.175, -59.795, 101.533, 200.777, 43.658, -195.349]
  MoveL 1288 to (-1100, 500, 50) mm, rotated rx 180 ry 0 rz 90 deg; joints [14.577, -61.583, 104.492, 200.904, 44.858, -195.15]
  MoveL 1289 to (-1100, 500, -0.5) mm, rotated rx -180 ry 0 rz 90 deg; joints [14.577, -59.696, 104.796, 200.159, 46.91, -194.079]
  MoveL 1290 to (-1100, 500, 50) mm, rotated rx 180 ry 0 rz 90 deg; joints [14.577, -61.583, 104.492, 200.904, 44.858, -195.15]
  MoveL 1291 to (-1100, 550, 50) mm, rotated rx 180 ry 0 rz 90 deg; joints [15.001, -63.36, 107.389, 201.084, 46.014, -194.99]
  MoveL 1292 to (-1100, 550, -0.5) mm, rotated rx -180 ry 0 rz 90 deg; joints [15.001, -61.404, 107.698, 200.339, 48.133, -193.896]
  MoveL 1293 to (-1100, 550, 50) mm, rotated rx 180 ry 0 rz 90 deg; joints [15.001, -63.36, 107.389, 201.084, 46.014, -194.99]
  MoveL 1294 to (-1100, 600, 50) mm, rotated rx -180 ry 0 rz 90 deg; joints [15.45, -65.128, 110.228, 201.315, 47.127, -194.867]
  MoveL 1295 to (-1100, 600, -0.5) mm, rotated rx 180 ry 0 rz 90 deg; joints [15.45, -63.1, 110.543, 200.566, 49.317, -193.744]
  MoveL 1296 to (-1100, 600, 50) mm, rotated rx -180 ry 0 rz 90 deg; joints [15.45, -65.128, 110.228, 201.315, 47.127, -194.867]
  MoveL 1297 to (-1100, 650, 50) mm, rotated rx -180 ry 0 rz 90 deg; joints [15.926, -66.894, 113.013, 201.598, 48.198, -194.782]
  MoveL 1298 to (-1100, 650, -0.5) mm, rotated rx -180 ry 0 rz 90 deg; joints [15.926, -64.787, 113.335, 200.842, 50.462, -193.623]
  MoveL 1299 to (-1100, 650, 50) mm, rotated rx -180 ry 0 rz 90 deg; joints [15.926, -66.894, 113.013, 201.598, 48.198, -194.782]
  MoveL 1300 to (-1100, 700, 50) mm, rotated rx 180 ry 0 rz 90 deg; joints [16.431, -68.661, 115.747, 201.933, 49.224, -194.734]
  MoveL 1301 to (-1100, 700, -0.5) mm, rotated rx -180 ry 0 rz 90 deg; joints [16.431, -66.471, 116.076, 201.167, 51.568, -193.533]
  MoveL 1302 to (-1100, 700, 50) mm, rotated rx 180 ry 0 rz 90 deg; joints [16.431, -68.661, 115.747, 201.933, 49.224, -194.734]
  MoveL 1303 to (-1100, 750, 50) mm, rotated rx -180 ry 0 rz 90 deg; joints [16.969, -70.434, 118.433, 202.323, 50.207, -194.724]
  MoveL 1304 to (-1100, 750, -0.5) mm, rotated rx 180 ry 0 rz 90 deg; joints [16.969, -68.154, 118.771, 201.543, 52.636, -193.473]
  MoveL 1305 to (-1100, 750, 50) mm, rotated rx -180 ry 0 rz 90 deg; joints [16.969, -70.434, 118.433, 202.323, 50.207, -194.724]
  MoveL 1306 to (-1100, 800, 50) mm, rotated rx -180 ry 0 rz 90 deg; joints [17.541, -72.217, 121.074, 202.77, 51.145, -194.753]
  MoveL 1307 to (-1100, 800, -0.5) mm, rotated rx -180 ry 0 rz 90 deg; joints [17.541, -69.842, 121.422, 201.971, 53.664, -193.444]
  MoveL 1308 to (-1100, 800, 50) mm, rotated rx -180 ry 0 rz 90 deg; joints [17.541, -72.217, 121.074, 202.77, 51.145, -194.753]
  MoveL 1309 to (-1100, 850, 50) mm, rotated rx -180 ry 0 rz 90 deg; joints [18.153, -74.016, 123.671, 203.277, 52.036, -194.823]
  MoveL 1310 to (-1100, 850, -0.5) mm, rotated rx -180 ry 0 rz 90 deg; joints [18.153, -71.537, 124.031, 202.456, 54.652, -193.448]
  MoveL 1311 to (-1100, 850, 50) mm, rotated rx -180 ry 0 rz 90 deg; joints [18.153, -74.016, 123.671, 203.277, 52.036, -194.823]
  MoveL 1312 to (-1100, 900, 50) mm, rotated rx 180 ry 0 rz 90 deg; joints [18.807, -75.836, 126.227, 203.848, 52.879, -194.937]
  MoveL 1313 to (-1100, 900, -0.5) mm, rotated rx -180 ry 0 rz 90 deg; joints [18.807, -73.245, 126.599, 202.999, 55.598, -193.486]
  MoveL 1314 to (-1100, 900, 50) mm, rotated rx 180 ry 0 rz 90 deg; joints [18.807, -75.836, 126.227, 203.848, 52.879, -194.937]
  MoveL 1315 to (-1100, 950, 50) mm, rotated rx -180 ry 0 rz 90 deg; joints [19.508, -77.683, 128.743, 204.488, 53.67, -195.101]
  MoveL 1316 to (-1100, 950, -0.5) mm, rotated rx -180 ry 0 rz 90 deg; joints [19.508, -74.971, 129.129, 203.607, 56.499, -193.562]
  MoveL 1317 to (-1100, 950, 50) mm, rotated rx -180 ry 0 rz 90 deg; joints [19.508, -77.683, 128.743, 204.488, 53.67, -195.101]
  MoveL 1318 to (-1100, 1000, 50) mm, rotated rx -180 ry 0 rz 90 deg; joints [20.26, -79.565, 131.219, 205.204, 54.408, -195.319]
  MoveL 1319 to (-1100, 1000, -0.5) mm, rotated rx -180 ry 0 rz 90 deg; joints [20.26, -76.721, 131.621, 204.284, 57.355, -193.679]
  MoveL 1320 to (-1100, 1000, 50) mm, rotated rx -180 ry 0 rz 90 deg; joints [20.26, -79.565, 131.219, 205.204, 54.408, -195.319]
  MoveL 1321 to (-1100, 1050, 50) mm, rotated rx -180 ry 0 rz 90 deg; joints [21.071, -81.488, 133.657, 206.004, 55.088, -195.599]
  MoveL 1322 to (-1100, 1050, -0.5) mm, rotated rx -180 ry 0 rz 90 deg; joints [21.071, -78.501, 134.076, 205.037, 58.161, -193.842]
  MoveL 1323 to (-1100, 1050, 50) mm, rotated rx -180 ry 0 rz 90 deg; joints [21.071, -81.488, 133.657, 206.004, 55.088, -195.599]
  MoveL 1324 to (-1100, 1100, 50) mm, rotated rx -180 ry 0 rz 90 deg; joints [21.946, -83.463, 136.057, 206.896, 55.706, -195.95]
  MoveL 1325 to (-1100, 1100, -0.5) mm, rotated rx 180 ry 0 rz 90 deg; joints [21.946, -80.319, 136.494, 205.874, 58.915, -194.059]
  MoveL 1326 to (-1100, 1100, 50) mm, rotated rx -180 ry 0 rz 90 deg; joints [21.946, -83.463, 136.057, 206.896, 55.706, -195.95]
  MoveL 1327 to (-1100, 1150, 50) mm, rotated rx -180 ry 0 rz 90 deg; joints [22.893, -85.499, 138.417, 207.892, 56.257, -196.384]
  MoveL 1328 to (-1100, 1150, -0.5) mm, rotated rx -180 ry 0 rz 90 deg; joints [22.893, -82.182, 138.876, 206.805, 59.611, -194.337]
  MoveL 1329 to (-1100, 1150, 50) mm, rotated rx -180 ry 0 rz 90 deg; joints [22.893, -85.499, 138.417, 207.892, 56.257, -196.384]
  MoveL 1330 to (-1100, 1200, 50) mm, rotated rx -180 ry 0 rz 90 deg; joints [23.92, -87.608, 140.738, 209.006, 56.738, -196.914]
  MoveL 1331 to (-1100, 1200, -0.5) mm, rotated rx -180 ry 0 rz 90 deg; joints [23.92, -84.103, 141.222, 207.841, 60.246, -194.688]
  MoveL 1332 to (-1100, 1200, 50) mm, rotated rx -180 ry 0 rz 90 deg; joints [23.92, -87.608, 140.738, 209.006, 56.738, -196.914]
  MoveL 1333 to (-1100, 1250, 50) mm, rotated rx -180 ry 0 rz 90 deg; joints [25.037, -89.805, 143.018, 210.252, 57.141, -197.56]
  MoveL 1334 to (-1100, 1250, -0.5) mm, rotated rx 180 ry 0 rz 90 deg; joints [25.037, -86.092, 143.529, 208.996, 60.813, -195.124]
  MoveL 1335 to (-1100, 1250, 50) mm, rotated rx -180 ry 0 rz 90 deg; joints [25.037, -89.805, 143.018, 210.252, 57.141, -197.56]
  MoveL 1336 to (-1100, 1300, 50) mm, rotated rx -180 ry 0 rz 90 deg; joints [26.256, -92.106, 145.255, 211.651, 57.462, -198.344]
  MoveL 1337 to (-1100, 1300, -0.5) mm, rotated rx 180 ry 0 rz 90 deg; joints [26.256, -88.165, 145.797, 210.285, 61.307, -195.663]
  MoveL 1338 to (-1100, 1300, 50) mm, rotated rx -180 ry 0 rz 90 deg; joints [26.256, -92.106, 145.255, 211.651, 57.462, -198.344]
  MoveL 1339 to (-1100, 1350, 50) mm, rotated rx -180 ry 0 rz 90 deg; joints [27.59, -94.532, 147.446, 213.227, 57.694, -199.295]
  MoveL 1340 to (-1100, 1350, -0.5) mm, rotated rx 180 ry 0 rz 90 deg; joints [27.59, -90.338, 148.024, 211.729, 61.721, -196.327]
  MoveL 1341 to (-1100, 1350, 50) mm, rotated rx -180 ry 0 rz 90 deg; joints [27.59, -94.532, 147.446, 213.227, 57.694, -199.295]
  MoveL 1342 to (-1170, 50, 50) mm, rotated rx 180 ry 0 rz 90 deg; joints [13.392, -43.771, 73.525, 205.63, 32.376, -202.057]
  MoveL 1343 to (-1170, 50, -0.5) mm, rotated rx -180 ry 0 rz 90 deg; joints [13.392, -42.373, 73.826, 204.527, 33.915, -200.74]
  MoveL 1344 to (-1170, 50, 50) mm, rotated rx 180 ry 0 rz 90 deg; joints [13.392, -43.771, 73.525, 205.63, 32.376, -202.057]
  MoveL 1345 to (-1170, 100, 50) mm, rotated rx -180 ry 0 rz 90 deg; joints [13.701, -45.863, 77.303, 205.05, 34.014, -201.176]
  MoveL 1346 to (-1170, 100, -0.5) mm, rotated rx -180 ry 0 rz 90 deg; joints [13.701, -44.421, 77.6, 204.012, 35.595, -199.912]
  MoveL 1347 to (-1170, 100, 50) mm, rotated rx -180 ry 0 rz 90 deg; joints [13.701, -45.863, 77.303, 205.05, 34.014, -201.176]
  MoveL 1348 to (-1170, 150, 50) mm, rotated rx 180 ry 0 rz 90 deg; joints [14.023, -47.888, 80.931, 204.609, 35.583, -200.431]
  MoveL 1349 to (-1170, 150, -0.5) mm, rotated rx 180 ry 0 rz 90 deg; joints [14.023, -46.402, 81.225, 203.623, 37.208, -199.205]
  MoveL 1350 to (-1170, 150, 50) mm, rotated rx 180 ry 0 rz 90 deg; joints [14.023, -47.888, 80.931, 204.609, 35.583, -200.431]
  MoveL 1351 to (-1170, 200, 50) mm, rotated rx 180 ry 0 rz 90 deg; joints [14.361, -49.856, 84.428, 204.284, 37.09, -199.794]
  MoveL 1352 to (-1170, 200, -0.5) mm, rotated rx -180 ry 0 rz 90 deg; joints [14.361, -48.323, 84.72, 203.339, 38.76, -198.596]
  MoveL 1353 to (-1170, 200, 50) mm, rotated rx 180 ry 0 rz 90 deg; joints [14.361, -49.856, 84.428, 204.284, 37.09, -199.794]
  MoveL 1354 to (-1170, 250, 50) mm, rotated rx 180 ry 0 rz 90 deg; joints [14.715, -51.776, 87.808, 204.058, 38.541, -199.249]
  MoveL 1355 to (-1170, 250, -0.5) mm, rotated rx 180 ry 0 rz 90 deg; joints [14.715, -50.195, 88.1, 203.145, 40.257, -198.068]
  MoveL 1356 to (-1170, 250, 50) mm, rotated rx 180 ry 0 rz 90 deg; joints [14.715, -51.776, 87.808, 204.058, 38.541, -199.249]
  MoveL 1357 to (-1170, 300, 50) mm, rotated rx -180 ry 0 rz 90 deg; joints [15.086, -53.656, 91.085, 203.918, 39.938, -198.781]
  MoveL 1358 to (-1170, 300, -0.5) mm, rotated rx 180 ry 0 rz 90 deg; joints [15.086, -52.025, 91.377, 203.031, 41.703, -197.609]
  MoveL 1359 to (-1170, 300, 50) mm, rotated rx -180 ry 0 rz 90 deg; joints [15.086, -53.656, 91.085, 203.918, 39.938, -198.781]
  MoveL 1360 to (-1170, 350, 50) mm, rotated rx -180 ry 0 rz 90 deg; joints [15.476, -55.502, 94.269, 203.854, 41.286, -198.38]
  MoveL 1361 to (-1170, 350, -0.5) mm, rotated rx -180 ry 0 rz 90 deg; joints [15.476, -53.817, 94.563, 202.986, 43.101, -197.209]
  MoveL 1362 to (-1170, 350, 50) mm, rotated rx -180 ry 0 rz 90 deg; joints [15.476, -55.502, 94.269, 203.854, 41.286, -198.38]
  MoveL 1363 to (-1170, 400, 50) mm, rotated rx 180 ry 0 rz 90 deg; joints [15.886, -57.318, 97.369, 203.859, 42.588, -198.037]
  MoveL 1364 to (-1170, 400, -0.5) mm, rotated rx 180 ry 0 rz 90 deg; joints [15.886, -55.578, 97.664, 203.007, 44.456, -196.861]
  MoveL 1365 to (-1170, 400, 50) mm, rotated rx 180 ry 0 rz 90 deg; joints [15.886, -57.318, 97.369, 203.859, 42.588, -198.037]
  MoveL 1366 to (-1170, 450, 50) mm, rotated rx 180 ry 0 rz 90 deg; joints [16.318, -59.112, 100.391, 203.93, 43.844, -197.747]
  MoveL 1367 to (-1170, 450, -0.5) mm, rotated rx 180 ry 0 rz 90 deg; joints [16.318, -57.312, 100.69, 203.087, 45.768, -196.56]
  MoveL 1368 to (-1170, 450, 50) mm, rotated rx 180 ry 0 rz 90 deg; joints [16.318, -59.112, 100.391, 203.93, 43.844, -197.747]
  MoveL 1369 to (-1170, 500, 50) mm, rotated rx -180 ry 0 rz 90 deg; joints [16.774, -60.886, 103.343, 204.062, 45.058, -197.506]
  MoveL 1370 to (-1170, 500, -0.5) mm, rotated rx 180 ry 0 rz 90 deg; joints [16.774, -59.024, 103.646, 203.225, 47.041, -196.3]
  MoveL 1371 to (-1170, 500, 50) mm, rotated rx -180 ry 0 rz 90 deg; joints [16.774, -60.886, 103.343, 204.062, 45.058, -197.506]
  MoveL 1372 to (-1170, 550, 50) mm, rotated rx -180 ry 0 rz 90 deg; joints [17.255, -62.646, 106.23, 204.252, 46.231, -197.31]
  MoveL 1373 to (-1170, 550, -0.5) mm, rotated rx -180 ry 0 rz 90 deg; joints [17.255, -60.718, 106.537, 203.417, 48.275, -196.08]
  MoveL 1374 to (-1170, 550, 50) mm, rotated rx -180 ry 0 rz 90 deg; joints [17.255, -62.646, 106.23, 204.252, 46.231, -197.31]
  MoveL 1375 to (-1170, 600, 50) mm, rotated rx -180 ry 0 rz 90 deg; joints [17.763, -64.395, 109.057, 204.501, 47.362, -197.156]
  MoveL 1376 to (-1170, 600, -0.5) mm, rotated rx 180 ry 0 rz 90 deg; joints [17.763, -62.397, 109.369, 203.664, 49.472, -195.895]
  MoveL 1377 to (-1170, 600, 50) mm, rotated rx -180 ry 0 rz 90 deg; joints [17.763, -64.395, 109.057, 204.501, 47.362, -197.156]
  MoveL 1378 to (-1170, 650, 50) mm, rotated rx 180 ry 0 rz 90 deg; joints [18.301, -66.138, 111.826, 204.807, 48.453, -197.043]
  MoveL 1379 to (-1170, 650, -0.5) mm, rotated rx -180 ry 0 rz 90 deg; joints [18.301, -64.065, 112.145, 203.965, 50.632, -195.745]
  MoveL 1380 to (-1170, 650, 50) mm, rotated rx 180 ry 0 rz 90 deg; joints [18.301, -66.138, 111.826, 204.807, 48.453, -197.043]
  MoveL 1381 to (-1170, 700, 50) mm, rotated rx -180 ry 0 rz 90 deg; joints [18.872, -67.879, 114.543, 205.172, 49.505, -196.971]
  MoveL 1382 to (-1170, 700, -0.5) mm, rotated rx -180 ry 0 rz 90 deg; joints [18.872, -65.726, 114.869, 204.32, 51.756, -195.629]
  MoveL 1383 to (-1170, 700, 50) mm, rotated rx -180 ry 0 rz 90 deg; joints [18.872, -67.879, 114.543, 205.172, 49.505, -196.971]
  MoveL 1384 to (-1170, 750, 50) mm, rotated rx 180 ry 0 rz 90 deg; joints [19.477, -69.622, 117.209, 205.596, 50.516, -196.941]
  MoveL 1385 to (-1170, 750, -0.5) mm, rotated rx -180 ry 0 rz 90 deg; joints [19.477, -67.384, 117.544, 204.731, 52.844, -195.547]
  MoveL 1386 to (-1170, 750, 50) mm, rotated rx 180 ry 0 rz 90 deg; joints [19.477, -69.622, 117.209, 205.596, 50.516, -196.941]
  MoveL 1387 to (-1170, 800, 50) mm, rotated rx -180 ry 0 rz 90 deg; joints [20.122, -71.371, 119.828, 206.082, 51.487, -196.952]
  MoveL 1388 to (-1170, 800, -0.5) mm, rotated rx 180 ry 0 rz 90 deg; joints [20.122, -69.042, 120.172, 205.201, 53.896, -195.498]
  MoveL 1389 to (-1170, 800, 50) mm, rotated rx -180 ry 0 rz 90 deg; joints [20.122, -71.371, 119.828, 206.082, 51.487, -196.952]
  MoveL 1390 to (-1170, 850, 50) mm, rotated rx 180 ry 0 rz 90 deg; joints [20.808, -73.13, 122.401, 206.633, 52.416, -197.007]
  MoveL 1391 to (-1170, 850, -0.5) mm, rotated rx 180 ry 0 rz 90 deg; joints [20.808, -70.703, 122.755, 205.731, 54.912, -195.484]
  MoveL 1392 to (-1170, 850, 50) mm, rotated rx 180 ry 0 rz 90 deg; joints [20.808, -73.13, 122.401, 206.633, 52.416, -197.007]
  MoveL 1393 to (-1170, 900, 50) mm, rotated rx 180 ry 0 rz 90 deg; joints [21.541, -74.905, 124.93, 207.253, 53.302, -197.11]
  MoveL 1394 to (-1170, 900, -0.5) mm, rotated rx 180 ry 0 rz 90 deg; joints [21.541, -72.373, 125.295, 206.325, 55.89, -195.507]
  MoveL 1395 to (-1170, 900, 50) mm, rotated rx 180 ry 0 rz 90 deg; joints [21.541, -74.905, 124.93, 207.253, 53.302, -197.11]
  MoveL 1396 to (-1170, 950, 50) mm, rotated rx 180 ry 0 rz 90 deg; joints [22.324, -76.701, 127.415, 207.947, 54.146, -197.262]
  MoveL 1397 to (-1170, 950, -0.5) mm, rotated rx 180 ry 0 rz 90 deg; joints [22.324, -74.054, 127.793, 206.988, 56.83, -195.569]
  MoveL 1398 to (-1170, 950, 50) mm, rotated rx 180 ry 0 rz 90 deg; joints [22.324, -76.701, 127.415, 207.947, 54.146, -197.262]
  MoveL 1399 to (-1170, 1000, 50) mm, rotated rx -180 ry 0 rz 90 deg; joints [23.164, -78.522, 129.858, 208.721, 54.943, -197.471]
  MoveL 1400 to (-1170, 1000, -0.5) mm, rotated rx 180 ry 0 rz 90 deg; joints [23.164, -75.753, 130.251, 207.724, 57.73, -195.674]
  MoveL 1401 to (-1170, 1000, 50) mm, rotated rx -180 ry 0 rz 90 deg; joints [23.164, -78.522, 129.858, 208.721, 54.943, -197.471]
  MoveL 1402 to (-1170, 1050, 50) mm, rotated rx 180 ry 0 rz 90 deg; joints [24.065, -80.377, 132.26, 209.58, 55.694, -197.741]
  MoveL 1403 to (-1170, 1050, -0.5) mm, rotated rx 180 ry 0 rz 90 deg; joints [24.065, -77.473, 132.668, 208.541, 58.589, -195.826]
  MoveL 1404 to (-1170, 1050, 50) mm, rotated rx 180 ry 0 rz 90 deg; joints [24.065, -80.377, 132.26, 209.58, 55.694, -197.741]
  MoveL 1405 to (-1170, 1100, 50) mm, rotated rx -180 ry 0 rz 90 deg; joints [25.034, -82.27, 134.62, 210.535, 56.396, -198.08]
  MoveL 1406 to (-1170, 1100, -0.5) mm, rotated rx 180 ry 0 rz 90 deg; joints [25.034, -79.222, 135.046, 209.445, 59.405, -196.03]
  MoveL 1407 to (-1170, 1100, 50) mm, rotated rx -180 ry 0 rz 90 deg; joints [25.034, -82.27, 134.62, 210.535, 56.396, -198.08]
  MoveL 1408 to (-1170, 1150, 50) mm, rotated rx -180 ry 0 rz 90 deg; joints [26.079, -84.211, 136.937, 211.594, 57.046, -198.499]
  MoveL 1409 to (-1170, 1150, -0.5) mm, rotated rx 180 ry 0 rz 90 deg; joints [26.079, -81.005, 137.383, 210.446, 60.176, -196.295]
  MoveL 1410 to (-1170, 1150, 50) mm, rotated rx -180 ry 0 rz 90 deg; joints [26.079, -84.211, 136.937, 211.594, 57.046, -198.499]
  MoveL 1411 to (-1170, 1200, 50) mm, rotated rx 180 ry 0 rz 90 deg; joints [27.208, -86.208, 139.212, 212.77, 57.644, -199.009]
  MoveL 1412 to (-1170, 1200, -0.5) mm, rotated rx 180 ry 0 rz 90 deg; joints [27.208, -82.83, 139.679, 211.552, 60.9, -196.627]
  MoveL 1413 to (-1170, 1200, 50) mm, rotated rx 180 ry 0 rz 90 deg; joints [27.208, -86.208, 139.212, 212.77, 57.644, -199.009]
  MoveL 1414 to (-1170, 1250, 50) mm, rotated rx 180 ry 0 rz 90 deg; joints [28.431, -88.272, 141.442, 214.074, 58.187, -199.624]
  MoveL 1415 to (-1170, 1250, -0.5) mm, rotated rx -180 ry 0 rz 90 deg; joints [28.431, -84.705, 141.934, 212.777, 61.575, -197.04]
  MoveL 1416 to (-1170, 1250, 50) mm, rotated rx 180 ry 0 rz 90 deg; joints [28.431, -88.272, 141.442, 214.074, 58.187, -199.624]
  MoveL 1417 to (-1170, 1300, 50) mm, rotated rx -180 ry 0 rz 90 deg; joints [29.759, -90.414, 143.625, 215.524, 58.675, -200.363]
  MoveL 1418 to (-1170, 1300, -0.5) mm, rotated rx -180 ry 0 rz 90 deg; joints [29.759, -86.642, 144.144, 214.133, 62.198, -197.546]
  MoveL 1419 to (-1170, 1300, 50) mm, rotated rx -180 ry 0 rz 90 deg; joints [29.759, -90.414, 143.625, 215.524, 58.675, -200.363]
  MoveL 1420 to (-1170, 1350, 50) mm, rotated rx -180 ry 0 rz 90 deg; joints [31.203, -92.647, 145.758, 217.137, 59.108, -201.247]
  MoveL 1421 to (-1170, 1350, -0.5) mm, rotated rx -180 ry 0 rz 90 deg; joints [31.203, -88.65, 146.309, 215.637, 62.769, -198.162]
  MoveL 1422 to (-1170, 1350, 50) mm, rotated rx -180 ry 0 rz 90 deg; joints [31.203, -92.647, 145.758, 217.137, 59.108, -201.247]
  MoveL 1423 to (-1240, 50, 50) mm, rotated rx 180 ry 0 rz 90 deg; joints [15.151, -43.01, 72.144, 209.081, 32.529, -205.123]
  MoveL 1424 to (-1240, 50, -0.5) mm, rotated rx 180 ry 0 rz 90 deg; joints [15.151, -41.627, 72.447, 207.857, 34.011, -203.658]
  MoveL 1425 to (-1240, 50, 50) mm, rotated rx 180 ry 0 rz 90 deg; joints [15.151, -43.01, 72.144, 209.081, 32.529, -205.123]
  MoveL 1426 to (-1240, 100, 50) mm, rotated rx -180 ry 0 rz 90 deg; joints [15.496, -45.111, 75.95, 208.406, 34.167, -204.108]
  MoveL 1427 to (-1240, 100, -0.5) mm, rotated rx 180 ry 0 rz 90 deg; joints [15.496, -43.686, 76.248, 207.254, 35.691, -202.703]
  MoveL 1428 to (-1240, 100, 50) mm, rotated rx -180 ry 0 rz 90 deg; joints [15.496, -45.111, 75.95, 208.406, 34.167, -204.108]
  MoveL 1429 to (-1240, 150, 50) mm, rotated rx 180 ry 0 rz 90 deg; joints [15.856, -47.141, 79.598, 207.891, 35.739, -203.248]
  MoveL 1430 to (-1240, 150, -0.5) mm, rotated rx 180 ry 0 rz 90 deg; joints [15.856, -45.672, 79.893, 206.796, 37.305, -201.887]
  MoveL 1431 to (-1240, 150, 50) mm, rotated rx 180 ry 0 rz 90 deg; joints [15.856, -47.141, 79.598, 207.891, 35.739, -203.248]
  MoveL 1432 to (-1240, 200, 50) mm, rotated rx 180 ry 0 rz 90 deg; joints [16.234, -49.112, 83.109, 207.507, 37.25, -202.514]
  MoveL 1433 to (-1240, 200, -0.5) mm, rotated rx -180 ry 0 rz 90 deg; joints [16.234, -47.597, 83.402, 206.459, 38.86, -201.183]
  MoveL 1434 to (-1240, 200, 50) mm, rotated rx 180 ry 0 rz 90 deg; joints [16.234, -49.112, 83.109, 207.507, 37.25, -202.514]
  MoveL 1435 to (-1240, 250, 50) mm, rotated rx 180 ry 0 rz 90 deg; joints [16.629, -51.031, 86.5, 207.235, 38.706, -201.883]
  MoveL 1436 to (-1240, 250, -0.5) mm, rotated rx 180 ry 0 rz 90 deg; joints [16.629, -49.469, 86.792, 206.225, 40.361, -200.574]
  MoveL 1437 to (-1240, 250, 50) mm, rotated rx 180 ry 0 rz 90 deg; joints [16.629, -51.031, 86.5, 207.235, 38.706, -201.883]
  MoveL 1438 to (-1240, 300, 50) mm, rotated rx 180 ry 0 rz 90 deg; joints [17.043, -52.906, 89.783, 207.06, 40.11, -201.341]
  MoveL 1439 to (-1240, 300, -0.5) mm, rotated rx -180 ry 0 rz 90 deg; joints [17.043, -51.296, 90.074, 206.08, 41.812, -200.042]
  MoveL 1440 to (-1240, 300, 50) mm, rotated rx 180 ry 0 rz 90 deg; joints [17.043, -52.906, 89.783, 207.06, 40.11, -201.341]
  MoveL 1441 to (-1240, 350, 50) mm, rotated rx 180 ry 0 rz 90 deg; joints [17.478, -54.745, 92.968, 206.972, 41.467, -200.874]
  MoveL 1442 to (-1240, 350, -0.5) mm, rotated rx 180 ry 0 rz 90 deg; joints [17.478, -53.083, 93.261, 206.015, 43.217, -199.579]
  MoveL 1443 to (-1240, 350, 50) mm, rotated rx 180 ry 0 rz 90 deg; joints [17.478, -54.745, 92.968, 206.972, 41.467, -200.874]
  MoveL 1444 to (-1240, 400, 50) mm, rotated rx -180 ry 0 rz 90 deg; joints [17.935, -56.553, 96.067, 206.962, 42.779, -200.474]
  MoveL 1445 to (-1240, 400, -0.5) mm, rotated rx 180 ry 0 rz 90 deg; joints [17.935, -54.836, 96.361, 206.022, 44.579, -199.175]
  MoveL 1446 to (-1240, 400, 50) mm, rotated rx -180 ry 0 rz 90 deg; joints [17.935, -56.553, 96.067, 206.962, 42.779, -200.474]
  MoveL 1447 to (-1240, 450, 50) mm, rotated rx -180 ry 0 rz 90 deg; joints [18.415, -58.334, 99.085, 207.024, 44.048, -200.133]
  MoveL 1448 to (-1240, 450, -0.5) mm, rotated rx 180 ry 0 rz 90 deg; joints [18.415, -56.56, 99.382, 206.097, 45.9, -198.823]
  MoveL 1449 to (-1240, 450, 50) mm, rotated rx -180 ry 0 rz 90 deg; joints [18.415, -58.334, 99.085, 207.024, 44.048, -200.133]
  MoveL 1450 to (-1240, 500, 50) mm, rotated rx 180 ry 0 rz 90 deg; joints [18.921, -60.093, 102.029, 207.154, 45.276, -199.847]
  MoveL 1451 to (-1240, 500, -0.5) mm, rotated rx -180 ry 0 rz 90 deg; joints [18.921, -58.26, 102.33, 206.236, 47.183, -198.519]
  MoveL 1452 to (-1240, 500, 50) mm, rotated rx 180 ry 0 rz 90 deg; joints [18.921, -60.093, 102.029, 207.154, 45.276, -199.847]
  MoveL 1453 to (-1240, 550, 50) mm, rotated rx 180 ry 0 rz 90 deg; joints [19.455, -61.835, 104.906, 207.35, 46.465, -199.61]
  MoveL 1454 to (-1240, 550, -0.5) mm, rotated rx 180 ry 0 rz 90 deg; joints [19.455, -59.938, 105.211, 206.436, 48.428, -198.258]
  MoveL 1455 to (-1240, 550, 50) mm, rotated rx 180 ry 0 rz 90 deg; joints [19.455, -61.835, 104.906, 207.35, 46.465, -199.61]
  MoveL 1456 to (-1240, 600, 50) mm, rotated rx 180 ry 0 rz 90 deg; joints [20.018, -63.564, 107.719, 207.609, 47.615, -199.42]
  MoveL 1457 to (-1240, 600, -0.5) mm, rotated rx -180 ry 0 rz 90 deg; joints [20.018, -61.6, 108.029, 206.695, 49.639, -198.037]
  MoveL 1458 to (-1240, 600, 50) mm, rotated rx 180 ry 0 rz 90 deg; joints [20.018, -63.564, 107.719, 207.609, 47.615, -199.42]
  MoveL 1459 to (-1240, 650, 50) mm, rotated rx -180 ry 0 rz 90 deg; joints [20.613, -65.283, 110.474, 207.931, 48.728, -199.276]
  MoveL 1460 to (-1240, 650, -0.5) mm, rotated rx 180 ry 0 rz 90 deg; joints [20.613, -63.247, 110.789, 207.014, 50.814, -197.855]
  MoveL 1461 to (-1240, 650, 50) mm, rotated rx -180 ry 0 rz 90 deg; joints [20.613, -65.283, 110.474, 207.931, 48.728, -199.276]
  MoveL 1462 to (-1240, 700, 50) mm, rotated rx 180 ry 0 rz 90 deg; joints [21.243, -66.996, 113.172, 208.317, 49.804, -199.175]
  MoveL 1463 to (-1240, 700, -0.5) mm, rotated rx 180 ry 0 rz 90 deg; joints [21.243, -64.885, 113.494, 207.392, 51.956, -197.71]
  MoveL 1464 to (-1240, 700, 50) mm, rotated rx 180 ry 0 rz 90 deg; joints [21.243, -66.996, 113.172, 208.317, 49.804, -199.175]
  MoveL 1465 to (-1240, 750, 50) mm, rotated rx 180 ry 0 rz 90 deg; joints [21.911, -68.707, 115.817, 208.766, 50.844, -199.119]
  MoveL 1466 to (-1240, 750, -0.5) mm, rotated rx -180 ry 0 rz 90 deg; joints [21.911, -66.515, 116.147, 207.83, 53.065, -197.6]
  MoveL 1467 to (-1240, 750, 50) mm, rotated rx 180 ry 0 rz 90 deg; joints [21.911, -68.707, 115.817, 208.766, 50.844, -199.119]
  MoveL 1468 to (-1240, 800, 50) mm, rotated rx 180 ry 0 rz 90 deg; joints [22.62, -70.42, 118.412, 209.282, 51.848, -199.106]
  MoveL 1469 to (-1240, 800, -0.5) mm, rotated rx 180 ry 0 rz 90 deg; joints [22.62, -68.142, 118.751, 208.331, 54.141, -197.527]
  MoveL 1470 to (-1240, 800, 50) mm, rotated rx 180 ry 0 rz 90 deg; joints [22.62, -70.42, 118.412, 209.282, 51.848, -199.106]
  MoveL 1471 to (-1240, 850, 50) mm, rotated rx -180 ry 0 rz 90 deg; joints [23.374, -72.139, 120.959, 209.866, 52.815, -199.14]
  MoveL 1472 to (-1240, 850, -0.5) mm, rotated rx 180 ry 0 rz 90 deg; joints [23.374, -69.768, 121.307, 208.896, 55.184, -197.491]
  MoveL 1473 to (-1240, 850, 50) mm, rotated rx -180 ry 0 rz 90 deg; joints [23.374, -72.139, 120.959, 209.866, 52.815, -199.14]
  MoveL 1474 to (-1240, 900, 50) mm, rotated rx 180 ry 0 rz 90 deg; joints [24.176, -73.867, 123.458, 210.522, 53.745, -199.221]
  MoveL 1475 to (-1240, 900, -0.5) mm, rotated rx -180 ry 0 rz 90 deg; joints [24.176, -71.396, 123.817, 209.529, 56.195, -197.493]
  MoveL 1476 to (-1240, 900, 50) mm, rotated rx 180 ry 0 rz 90 deg; joints [24.176, -73.867, 123.458, 210.522, 53.745, -199.221]
  MoveL 1477 to (-1240, 950, 50) mm, rotated rx 180 ry 0 rz 90 deg; joints [25.032, -75.608, 125.912, 211.255, 54.639, -199.353]
  MoveL 1478 to (-1240, 950, -0.5) mm, rotated rx -180 ry 0 rz 90 deg; joints [25.032, -73.032, 126.282, 210.235, 57.172, -197.535]
  MoveL 1479 to (-1240, 950, 50) mm, rotated rx 180 ry 0 rz 90 deg; joints [25.032, -75.608, 125.912, 211.255, 54.639, -199.353]
  MoveL 1480 to (-1240, 1000, 50) mm, rotated rx -180 ry 0 rz 90 deg; joints [25.946, -77.368, 128.32, 212.069, 55.495, -199.541]
  MoveL 1481 to (-1240, 1000, -0.5) mm, rotated rx 180 ry 0 rz 90 deg; joints [25.946, -74.677, 128.703, 211.016, 58.115, -197.619]
  MoveL 1482 to (-1240, 1000, 50) mm, rotated rx -180 ry 0 rz 90 deg; joints [25.946, -77.368, 128.32, 212.069, 55.495, -199.541]
  MoveL 1483 to (-1240, 1050, 50) mm, rotated rx -180 ry 0 rz 90 deg; joints [26.925, -79.151, 130.683, 212.97, 56.314, -199.788]
  MoveL 1484 to (-1240, 1050, -0.5) mm, rotated rx 180 ry 0 rz 90 deg; joints [26.925, -76.337, 131.081, 211.88, 59.025, -197.75]
  MoveL 1485 to (-1240, 1050, 50) mm, rotated rx -180 ry 0 rz 90 deg; joints [26.925, -79.151, 130.683, 212.97, 56.314, -199.788]
  MoveL 1486 to (-1240, 1100, 50) mm, rotated rx -180 ry 0 rz 90 deg; joints [27.974, -80.963, 133.001, 213.967, 57.094, -200.102]
  MoveL 1487 to (-1240, 1100, -0.5) mm, rotated rx -180 ry 0 rz 90 deg; joints [27.974, -78.016, 133.415, 212.833, 59.9, -197.932]
  MoveL 1488 to (-1240, 1100, 50) mm, rotated rx -180 ry 0 rz 90 deg; joints [27.974, -80.963, 133.001, 213.967, 57.094, -200.102]
  MoveL 1489 to (-1240, 1150, 50) mm, rotated rx 180 ry 0 rz 90 deg; joints [29.101, -82.809, 135.274, 215.066, 57.836, -200.489]
  MoveL 1490 to (-1240, 1150, -0.5) mm, rotated rx 180 ry 0 rz 90 deg; joints [29.101, -79.717, 135.705, 213.882, 60.741, -198.17]
  MoveL 1491 to (-1240, 1150, 50) mm, rotated rx 180 ry 0 rz 90 deg; joints [29.101, -82.809, 135.274, 215.066, 57.836, -200.489]
  MoveL 1492 to (-1240, 1200, 50) mm, rotated rx -180 ry 0 rz 90 deg; joints [30.314, -84.695, 137.499, 216.278, 58.541, -200.96]
  MoveL 1493 to (-1240, 1200, -0.5) mm, rotated rx -180 ry 0 rz 90 deg; joints [30.314, -81.448, 137.95, 215.036, 61.546, -198.472]
  MoveL 1494 to (-1240, 1200, 50) mm, rotated rx -180 ry 0 rz 90 deg; joints [30.314, -84.695, 137.499, 216.278, 58.541, -200.96]
  MoveL 1495 to (-1240, 1250, 50) mm, rotated rx 180 ry 0 rz 90 deg; joints [31.621, -86.629, 139.677, 217.613, 59.21, -201.524]
  MoveL 1496 to (-1240, 1250, -0.5) mm, rotated rx -180 ry 0 rz 90 deg; joints [31.621, -83.213, 140.149, 216.304, 62.317, -198.846]
  MoveL 1497 to (-1240, 1250, 50) mm, rotated rx 180 ry 0 rz 90 deg; joints [31.621, -86.629, 139.677, 217.613, 59.21, -201.524]
  MoveL 1498 to (-1240, 1300, 50) mm, rotated rx -180 ry 0 rz 90 deg; joints [33.033, -88.618, 141.803, 219.083, 59.843, -202.196]
  MoveL 1499 to (-1240, 1300, -0.5) mm, rotated rx 180 ry 0 rz 90 deg; joints [33.033, -85.019, 142.3, 217.699, 63.054, -199.301]
  MoveL 1500 to (-1240, 1300, 50) mm, rotated rx -180 ry 0 rz 90 deg; joints [33.033, -88.618, 141.803, 219.083, 59.843, -202.196]
  MoveL 1501 to (-1240, 1350, 50) mm, rotated rx -180 ry 0 rz 90 deg; joints [34.56, -90.67, 143.877, 220.701, 60.447, -202.99]
  MoveL 1502 to (-1240, 1350, -0.5) mm, rotated rx 180 ry 0 rz 90 deg; joints [34.56, -86.873, 144.4, 219.232, 63.759, -199.85]
  MoveL 1503 to (-1240, 1350, 50) mm, rotated rx -180 ry 0 rz 90 deg; joints [34.56, -90.67, 143.877, 220.701, 60.447, -202.99]
  MoveL 1504 to (-1240, 1400, 50) mm, rotated rx 180 ry 0 rz 90 deg; joints [36.216, -92.794, 145.894, 222.483, 61.025, -203.923]
  MoveL 1505 to (-1240, 1400, -0.5) mm, rotated rx 180 ry 0 rz 90 deg; joints [36.216, -88.782, 146.446, 220.917, 64.435, -200.507]
  MoveL 1506 to (-1240, 1400, 50) mm, rotated rx 180 ry 0 rz 90 deg; joints [36.216, -92.794, 145.894, 222.483, 61.025, -203.923]
  MoveL 1507 to (-1240, 1450, 50) mm, rotated rx 180 ry 0 rz 90 deg; joints [38.014, -95, 147.849, 224.442, 61.589, -205.014]
  MoveL 1508 to (-1240, 1450, -0.5) mm, rotated rx -180 ry 0 rz 90 deg; joints [38.014, -90.755, 148.434, 222.768, 65.087, -201.288]
  MoveL 1509 to (-1240, 1450, 50) mm, rotated rx 180 ry 0 rz 90 deg; joints [38.014, -95, 147.849, 224.442, 61.589, -205.014]
  MoveL 1510 to (-1310, 50, 50) mm, rotated rx 180 ry 0 rz 90 deg; joints [16.881, -42.146, 70.572, 212.517, 32.697, -208.212]
  MoveL 1511 to (-1310, 50, -0.5) mm, rotated rx -180 ry 0 rz 90 deg; joints [16.881, -40.78, 70.878, 211.179, 34.117, -206.61]
  MoveL 1512 to (-1310, 50, 50) mm, rotated rx 180 ry 0 rz 90 deg; joints [16.881, -42.146, 70.572, 212.517, 32.697, -208.212]
  MoveL 1513 to (-1310, 100, 50) mm, rotated rx -180 ry 0 rz 90 deg; joints [17.26, -44.26, 74.412, 211.74, 34.335, -207.058]
  MoveL 1514 to (-1310, 100, -0.5) mm, rotated rx 180 ry 0 rz 90 deg; joints [17.26, -42.852, 74.711, 210.483, 35.797, -205.522]
  MoveL 1515 to (-1310, 100, 50) mm, rotated rx -180 ry 0 rz 90 deg; joints [17.26, -44.26, 74.412, 211.74, 34.335, -207.058]
  MoveL 1516 to (-1310, 150, 50) mm, rotated rx 180 ry 0 rz 90 deg; joints [17.657, -46.298, 78.085, 211.143, 35.908, -206.079]
  MoveL 1517 to (-1310, 150, -0.5) mm, rotated rx 180 ry 0 rz 90 deg; joints [17.657, -44.847, 78.381, 209.951, 37.412, -204.592]
  MoveL 1518 to (-1310, 150, 50) mm, rotated rx 180 ry 0 rz 90 deg; joints [17.657, -46.298, 78.085, 211.143, 35.908, -206.079]
  MoveL 1519 to (-1310, 200, 50) mm, rotated rx -180 ry 0 rz 90 deg; joints [18.072, -48.271, 81.616, 210.695, 37.423, -205.242]
  MoveL 1520 to (-1310, 200, -0.5) mm, rotated rx -180 ry 0 rz 90 deg; joints [18.072, -46.777, 81.909, 209.554, 38.97, -203.79]
  MoveL 1521 to (-1310, 200, 50) mm, rotated rx -180 ry 0 rz 90 deg; joints [18.072, -48.271, 81.616, 210.695, 37.423, -205.242]
  MoveL 1522 to (-1310, 250, 50) mm, rotated rx -180 ry 0 rz 90 deg; joints [18.506, -50.191, 85.019, 210.372, 38.884, -204.522]
  MoveL 1523 to (-1310, 250, -0.5) mm, rotated rx 180 ry 0 rz 90 deg; joints [18.506, -48.65, 85.311, 209.274, 40.474, -203.095]
  MoveL 1524 to (-1310, 250, 50) mm, rotated rx -180 ry 0 rz 90 deg; joints [18.506, -50.191, 85.019, 210.372, 38.884, -204.522]
  MoveL 1525 to (-1310, 300, 50) mm, rotated rx -180 ry 0 rz 90 deg; joints [18.96, -52.063, 88.31, 210.158, 40.296, -203.901]
  MoveL 1526 to (-1310, 300, -0.5) mm, rotated rx -180 ry 0 rz 90 deg; joints [18.96, -50.475, 88.602, 209.093, 41.93, -202.488]
  MoveL 1527 to (-1310, 300, 50) mm, rotated rx -180 ry 0 rz 90 deg; joints [18.96, -52.063, 88.31, 210.158, 40.296, -203.901]
  MoveL 1528 to (-1310, 350, 50) mm, rotated rx -180 ry 0 rz 90 deg; joints [19.437, -53.895, 91.5, 210.04, 41.661, -203.366]
  MoveL 1529 to (-1310, 350, -0.5) mm, rotated rx -180 ry 0 rz 90 deg; joints [19.437, -52.257, 91.792, 209.002, 43.341, -201.958]
  MoveL 1530 to (-1310, 350, 50) mm, rotated rx -180 ry 0 rz 90 deg; joints [19.437, -53.895, 91.5, 210.04, 41.661, -203.366]
  MoveL 1531 to (-1310, 400, 50) mm, rotated rx -180 ry 0 rz 90 deg; joints [19.937, -55.693, 94.598, 210.009, 42.983, -202.905]
